// TIA Portal project "Project 3 Template_V15" (V15)

(* hardware
DEVICE "ET 200SP station_1"  ET 200SP-Station
   slot 0: "Rack_0"  Rack  6ES5 710-8MAx1
   slot 1: "PROJECT"  CPU 1512SP F-1 PN  6ES7 512-1SK01-0AB0  V1.8
   slot 2: "DC Input Card 1"  DI 8x24VDC HF  6ES7 131-6BF00-0CA0  V1.2
      slot 1: "DC Input Card 1"  DI 8x24VDC HF
   slot 3: "DC Input Card 2"  DI 8x24VDC HF  6ES7 131-6BF00-0CA0  V1.2
      slot 1: "DC Input Card 2"  DI 8x24VDC HF
   slot 4: "DC Output Card 1"  DQ 8x24VDC/0.5A HF  6ES7 132-6BF00-0CA0  V1.2
      slot 1: "DC Output Card 1"  DQ 8x24VDC/0.5A HF
   slot 5: "DC Output Card 2"  DQ 8x24VDC/0.5A HF  6ES7 132-6BF00-0CA0  V1.2
      slot 1: "DC Output Card 2"  DQ 8x24VDC/0.5A HF
   slot 6: "Analog Input Card 1"  AI 2xU/I 2,4-wire HS  6ES7 134-6HB00-0DA1  V1.1
      slot 1: "Analog Input Card 1"  AI 2xU/I 2,4-wire HS
   slot 7: "Analog Input Card 1_1"  AI 2xU/I 2,4-wire HS  6ES7 134-6HB00-0DA1  V1.1
      slot 1: "Analog Input Card 1_1"  AI 2xU/I 2,4-wire HS
   slot 8: "Analog Output Card"  AQ 2xU/I HS  6ES7 135-6HB00-0DA1  V1.1
      slot 1: "Analog Output Card"  AQ 2xU/I HS
   slot 9: "Server module_1"  Server module  6ES7 193-6PA00-0AA0  V1.0
      slot 1: "Server module_1"  Server module
   slot 127: "PROFINET BusAdapter CU"  BA 2xRJ45  6ES7 193-6AR00-0AA0  V0.0
      slot 32769: "Port_1"  6ES7 193-6AR00-0AA0
      slot 32770: "Port_2"  6ES7 193-6AR00-0AA0
DEVICE "GSD device_1"  GSD.Device.PN
   slot 0: "Rack"  Rail  V1.0
   slot 0: "WAGO"  750-377  V02.01.xx (03/04)
   slot 1: "75x-431 8DI_1"  75x-431
   slot 2: "75x-431 8DI_2"  75x-431
   slot 3: "75x-530(/0..-...) 8DO_1"  75x-530
   slot 4: "75x-530(/0..-...) 8DO_2"  75x-530
DEVICE "Visual Interface Simulator"  TP900 Comfort Portrait
   slot 0: "Visual Interface Simulator"  TP900 Comfort Portrait  6AV2 124-0JC01-0AX0  15.0.0.0
   slot 1: "HMI_RT_1"  TP900 Comfort Portrait  6AV2 124-0JC01-0AX0  15.0.0.0
   slot 5: "Visual Interface Simulator.IE_CP_1"  PROFINET Interface  15.0.0.0
      slot 1: "PROFINET Interface_1"  PROFINET Interface
         slot 1: "Port_1"  Port
         slot 2: "Port_2"  Port
   slot 7: "Visual Interface Simulator.MPI/DP_CP_1"  MPI/DP Interface  15.0.0.0
*)

// ===== PLC "PROJECT"  CPU 1512SP F-1 PN =====

VAR_GLOBAL   // PLC tag table "Default tag table"
   "Tag_1" AT %M1.0 : Bool;
   "INRange" AT %M1.4 : Bool;
   "Tag_3" AT %M13.1 : Bool;
   "Tag_4" AT %M9.0 : Bool;
   "Tag_6" AT %M7.1 : Bool;
   "FaultDetected" AT %M14.1 : Bool;
END_VAR

VAR_GLOBAL   // PLC tag table "R99_SIM Tags"
   "QB0" AT %QB0 : Byte;
   "IB0" AT %IB0 : Byte;
   "QB1" AT %QB1 : Byte;
   "QB70" AT %QB70 : Byte;
   "QB71" AT %QB71 : Byte;
   "IB1" AT %IB1 : Byte;
   "IB70" AT %IB70 : Byte;
   "IB71" AT %IB71 : Byte;
   "IW2" AT %IW2 : Int;
END_VAR

VAR_GLOBAL CONSTANT   // PLC tag table "R99_SIM Tags"
   "None(1)" : Pip := 65535;
   "Automatic update(1)" : Pip := 0;
   "PIP 1(1)" : Pip := 1;
   "PIP 2(1)" : Pip := 2;
   "PIP 3(1)" : Pip := 3;
   "PIP 4(1)" : Pip := 4;
   "PIP 5(1)" : Pip := 5;
   "PIP 6(1)" : Pip := 6;
   "PIP 7(1)" : Pip := 7;
   "PIP 8(1)" : Pip := 8;
   "PIP 9(1)" : Pip := 9;
   "PIP 10(1)" : Pip := 10;
   "PIP 11(1)" : Pip := 11;
   "PIP 12(1)" : Pip := 12;
   "PIP 13(1)" : Pip := 13;
   "PIP 14(1)" : Pip := 14;
   "PIP 15(1)" : Pip := 15;
   "PIP 16(1)" : Pip := 16;
   "PIP 17(1)" : Pip := 17;
   "PIP 18(1)" : Pip := 18;
   "PIP 19(1)" : Pip := 19;
   "PIP 20(1)" : Pip := 20;
   "PIP 21(1)" : Pip := 21;
   "PIP 22(1)" : Pip := 22;
   "PIP 23(1)" : Pip := 23;
   "PIP 24(1)" : Pip := 24;
   "PIP 25(1)" : Pip := 25;
   "PIP 26(1)" : Pip := 26;
   "PIP 27(1)" : Pip := 27;
   "PIP 28(1)" : Pip := 28;
   "PIP 29(1)" : Pip := 29;
   "PIP 30(1)" : Pip := 30;
   "PIP 31(1)" : Pip := 31;
   "PIP OB Servo(1)" : Pip := 32768;
   "Local~MC(1)" : Hw_SubModule := 51;
   "Local~Common(1)" : Hw_SubModule := 50;
   "Local~Device(1)" : Hw_Device := 32;
   "Local~Configuration(1)" : Hw_SubModule := 33;
   "Local~Exec(1)" : Hw_SubModule := 52;
   "Local(1)" : Hw_SubModule := 49;
   "Local~FExec(1)" : Hw_SubModule := 55;
   "Local~PROFINET_interface_1(1)" : Hw_Interface := 64;
   "Local~PROFINET_interface_1~Port_3(1)" : Hw_Interface := 67;
   "Local~PROFINET_interface_1~Port_1(1)" : Hw_Interface := 65;
   "Local~PROFINET_interface_1~Port_2(1)" : Hw_Interface := 66;
   "OB_Main(1)" : OB_PCYCLE := 1;
   "Local~DC_Input_Card_1_1(1)" : Hw_SubModule := 257;
   "Local~DC_Input_Card_2_1(1)" : Hw_SubModule := 258;
   "Local~DC_Output_Card_1_1(1)" : Hw_SubModule := 259;
   "Local~DC_Output_Card_2_1(1)" : Hw_SubModule := 260;
   "Local~Analog_Input_Card_1_1(1)" : Hw_SubModule := 261;
   "Local~Analog_Output_Card_1(1)" : Hw_SubModule := 263;
   "Local~Analog_Input_Card_1_1_2(1)" : Hw_SubModule := 262;
   "Local~PROFINET_IO-System(1)" : Hw_IoSystem := 264;
   "WAGO~Proxy(1)" : Hw_SubModule := 268;
   "WAGO~IODevice(1)" : Hw_Device := 266;
   "WAGO~Interface(1)" : Hw_Interface := 269;
   "WAGO~Interface~Port_1(1)" : Hw_Interface := 270;
   "WAGO~Interface~Port_2(1)" : Hw_Interface := 271;
   "WAGO~Head(1)" : Hw_SubModule := 272;
   "8DI~DI(2)" : Hw_SubModule := 273;
   "8DI~DI(3)" : Hw_SubModule := 274;
   "8DO~DO(2)" : Hw_SubModule := 275;
   "8DO~DO(3)" : Hw_SubModule := 276;
END_VAR

VAR_GLOBAL   // PLC tag table "project M File tag"
   "PNPExt" AT %Q70.0 : Bool;
   "PNPRet" AT %Q70.1 : Bool;
   "PNPRaise" AT %Q70.2 : Bool;
   "PNPlower" AT %Q70.3 : Bool;
   "PNPGrip" AT %Q70.4 : Bool;
   "ConEXT" AT %Q70.5 : Bool;
   "ConvRun" AT %Q70.6 : Bool;
   "extendPNP" AT %I70.0 : Bool;
   "retractPNP" AT %I70.1 : Bool;
   "raised" AT %I70.2 : Bool;
   "lower" AT %I70.3 : Bool;
   "Tag_5" AT %I70.4 : Bool;
   "convRet" AT %I70.5 : Bool;
   "partAtPickUp" AT %I70.6 : Bool;
   "StartPB" AT %I0.0 : Bool;
   "StopPB" AT %I0.1 : Bool;
   "PBA" AT %I0.2 : Bool;
   "PBB" AT %I0.3 : Bool;
   "SSA" AT %I0.4 : Bool;
   "MCR" AT %I0.5 : Bool;
   "EStopPB" AT %I0.6 : Bool;
   "GateSwitch" AT %I0.7 : Bool;
   "StartLight" AT %Q0.0 : Bool;
   "Tag_2" AT %Q0.1 : Bool;
   "LTA" AT %Q0.2 : Bool;
   "LTB" AT %Q0.3 : Bool;
END_VAR

TYPE "TPBool"
VERSION : 0.1
   STRUCT
      PB : Bool;
      LT : Bool;
   END_STRUCT;
END_TYPE

TYPE "TouchPanelPLC"
VERSION : 0.1
   STRUCT
      INT1 : Int;
      INT2 : Int;
      INT3 : Int;
      INT4 : Int;
      REAL1 : Real;
      REAL2 : Real;
      REAL3 : Real;
      REAL4 : Real;
      GRAY : "TPBool";
      BLUE : "TPBool";
      GREEN : "TPBool";
      YELLOW : "TPBool";
      RED : "TPBool";
   END_STRUCT;
END_TYPE

TYPE "TouchPanel"
VERSION : 0.1
   STRUCT
      PLC : "TouchPanelPLC";
      Stn : "TouchPanelStn";
      Conv : "TouchPanelConv";
   END_STRUCT;
END_TYPE

TYPE "TPExtRet"
VERSION : 0.1
   STRUCT
      Ext : "TPBool";
      Ret : "TPBool";
   END_STRUCT;
END_TYPE

TYPE "TPRaiseLower"
VERSION : 0.1
   STRUCT
      Raise : "TPBool";
      Lower : "TPBool";
   END_STRUCT;
END_TYPE

TYPE "TPOnOff"
VERSION : 0.1
   STRUCT
      On : "TPBool";
      Off : "TPBool";
   END_STRUCT;
END_TYPE

TYPE "TouchPanelStn"
VERSION : 0.1
   STRUCT
      Auto : "TPBool";
      Manual : "TPBool";
      CycleStart : "TPBool";
      CycleStop : "TPBool";
      Lift : "TPRaiseLower";
      PartRelease : "TPOnOff";
      Reject : "TPExtRet";
      Divert : "TPExtRet";
      SendToRejectChute : "TPBool";
      SendToDivertChute : "TPBool";
      SendToConv : "TPBool";
      InsertPart : "TPBool";
      FaultReset : "TPBool";
   END_STRUCT;
END_TYPE

TYPE "TouchPanelConv"
VERSION : 0.1
   STRUCT
      TargetSpeed : Real;
      Fwd : "TPBool";
      Rev : "TPBool";
      Stop : "TPBool";
      FaultReset : "TPBool";
      RemCntl : "TPOnOff";
   END_STRUCT;
END_TYPE

TYPE "SIM_CylinderAnimation"
VERSION : 0.1
   STRUCT
      Animation : DInt;
      Max : DInt;
      Extend : "SIM_Cylinder";
      Retract : "SIM_Cylinder";
   END_STRUCT;
END_TYPE

TYPE "SIM_Cylinder"
VERSION : 0.1
   STRUCT
      ScanCount : DInt;
      "Timer" : IEC_TIMER;
      Output : Bool;
      Sensor : Bool;
   END_STRUCT;
END_TYPE

TYPE "SIM_PLC"
VERSION : 0.1
   STRUCT
      IB0 : Byte;
      IB1 : Byte;
      IB70 : Byte;
      IB71 : Byte;
      QB0 : Byte;
      QB1 : Byte;
      QB70 : Byte;
      QB71 : Byte;
      PowerOnPB : Bool;
      Lift : "SIM_CylinderAnimation";
      Reject : "SIM_CylinderAnimation";
      Divert : "SIM_CylinderAnimation";
      "5sPulse" : IEC_TIMER;
      PartRelease : Bool;
      IW2 : Int;
      Oneshots : "Numbers";
      RandomTimer : IEC_TIMER;
      CH0RampUP : IEC_TIMER;
      CH0ACC : Int;
      RandomTime : Int;
      NewPartDelay : IEC_TIMER;
      PartClearDelay : IEC_TIMER;
   END_STRUCT;
END_TYPE

TYPE "Numbers"
VERSION : 0.1
   STRUCT
      "0" : Bool;
      "1" : Bool;
      "2" : Bool;
      "3" : Bool;
      "4" : Bool;
      "5" : Bool;
      "6" : Bool;
      "7" : Bool;
      "8" : Bool;
      "9" : Bool;
      "10" : Bool;
      "11" : Bool;
      "12" : Bool;
      "13" : Bool;
      "14" : Bool;
      "15" : Bool;
   END_STRUCT;
END_TYPE

DATA_BLOCK "TP"   // DB1
{ S7_Optimized_Access := 'FALSE' }
VERSION : 0.1
BEGIN
   PLC.GRAY.PB := true;
END_DATA_BLOCK

DATA_BLOCK "SIM"   // DB2
{ S7_Optimized_Access := 'FALSE' }
VERSION : 0.1
BEGIN
   IB0 := 2#10000010;
   Lift.Retract.Sensor := true;
   Reject.Retract.Sensor := true;
   Divert.Retract.Output := true;
   IB70 := 2#00000110;
END_DATA_BLOCK

DATA_BLOCK "project"   // DB3
{ S7_Optimized_Access := 'TRUE' }
VERSION : 0.1
   VAR
      RejectPartCount : Int;
      MaxWeight : Real;
      CycletimeREal : Real;
      cycletimeint : Int;
      PrevMaxWeight : Real;
      MaxWeigInt : Int;
   END_VAR
BEGIN
END_DATA_BLOCK

DATA_BLOCK "Project timers and counters"   // DB4
{ S7_Optimized_Access := 'TRUE' }
VERSION : 0.1
   VAR
      FaultTimer : IEC_TIMER;
      GoodPartCounters : IEC_COUNTER;
   END_VAR
   VAR RETAIN
      CycleTimer : IEC_TIMER;
   END_VAR
   VAR
      RetractionDelayTimer : IEC_TIMER;
      tptimer : IEC_TIMER;
      tofftimer : IEC_TIMER;
      extendGreenLt : IEC_TIMER;
   END_VAR
BEGIN
END_DATA_BLOCK

DATA_BLOCK "String Variables"   // DB12
{ S7_Optimized_Access := 'TRUE' }
VERSION : 0.1
   VAR RETAIN
      REAL1_TEXT : String := 'Real weight';
      REAL2_TEXT : String := 'curr weight';
      REAL3_TEXT : String := 'cycle time';
      REAL4_TEXT : String := 'Not used';
      INT1_TEXT : String := 'good part';
      INT2_TEXT : String := 'bad parts';
      INT3_TEXT : String := 'lower range';
      INT4_TEXT : String := 'higher range';
   END_VAR
BEGIN
END_DATA_BLOCK

FUNCTION "System Control" : Void   // FC1, LAD
{ S7_Optimized_Access := 'TRUE' }
VERSION : 0.1
// To Active cycle time, Press start PB , turn on MCR, the stop the it press PB
BEGIN

REGION Network 1
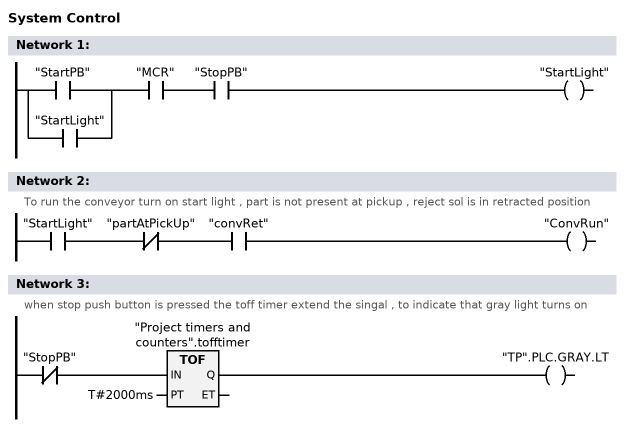
   RUNG wire#powerrail
      Contact( "StartPB" )
      wire#w1
      Contact( "MCR" )
      Contact( "StopPB" )
      Coil( "StartLight" )
   END_RUNG
   RUNG wire#powerrail
      Contact( "StartLight" )
   END_RUNG wire#w1
   // the same network as SCL:
   "StartLight" := ("StartPB" OR "StartLight") AND "MCR" AND "StopPB";
END_REGION

REGION Network 2
   // To run the conveyor turn on start light , part is not present at pickup , reject sol is in retracted position
   RUNG wire#powerrail
      Contact( "StartLight" )
      I_Contact( "partAtPickUp" )
      Contact( "convRet" )
      Coil( "ConvRun" )
   END_RUNG
   // the same network as SCL:
   "ConvRun" := "StartLight" AND NOT "partAtPickUp" AND "convRet";
END_REGION

REGION Network 3
   // when stop push button is pressed the toff timer extend the singal , to indicate that gray light turns on
   "Project timers and counters".tofftimer.TOF(IN := NOT "StopPB", PT := T#2000ms);
   "TP".PLC.GRAY.LT := "Project timers and counters".tofftimer.Q;
END_REGION
END_FUNCTION

FUNCTION "Weight Check Station Control" : Void   // FC2, LAD
{ S7_Optimized_Access := 'TRUE' }
VERSION : 0.1
   VAR_TEMP   // added for the SCL form of the ladder/FBD networks
      _w1 : Bool;
   END_VAR
BEGIN

REGION Network 1
   // To calculate the weight we need to convert the Analog value to the real weight in gms and displayed in real 1
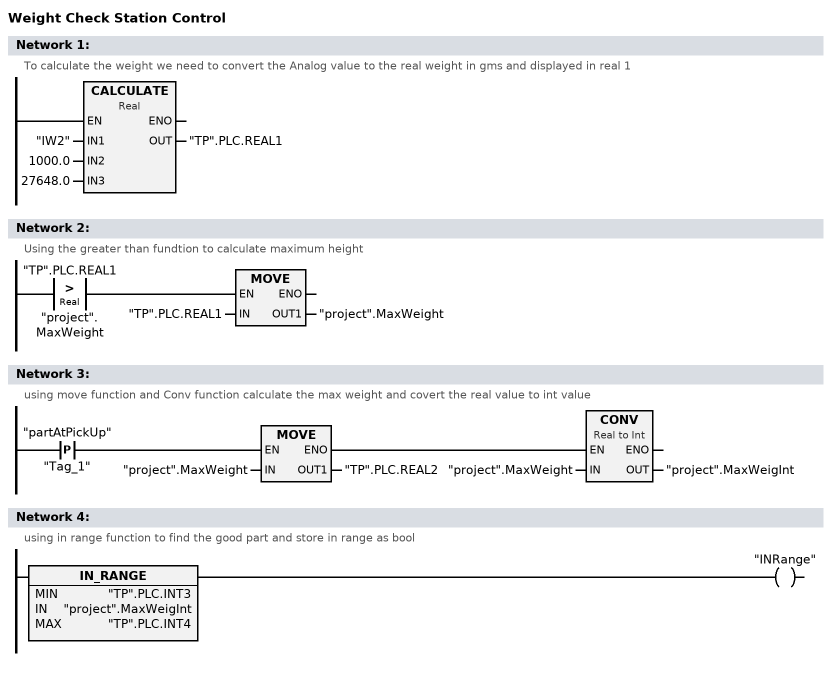
   RUNG wire#powerrail
      { S7_Templates := "SrcType := Real"; S7_Expression := "(IN2 / IN3) * IN1" } Calculate(in1 := "IW2", in2 := 1000.0, in3 := 27648.0, out => "TP".PLC.REAL1)
   END_RUNG
   // the same network as SCL:
   "TP".PLC.REAL1 := (1000.0 / 27648.0) * "IW2";
END_REGION

REGION Network 2
   // Using the greater than fundtion to calculate maximum height
   RUNG wire#powerrail
      { S7_Templates := "SrcType := Real" } GT_Contact(in1 := "TP".PLC.REAL1, in2 := "project".MaxWeight)
      Move(in := "TP".PLC.REAL1, out1 => "project".MaxWeight)
   END_RUNG
   // the same network as SCL:
   IF "TP".PLC.REAL1 > "project".MaxWeight THEN "project".MaxWeight := "TP".PLC.REAL1; END_IF;
END_REGION

REGION Network 3
   // using move function and Conv function calculate the max weight and covert the real value to int value
   RUNG wire#powerrail
      P_Contact(operand := "partAtPickUp", bit := "Tag_1")
      Move(in := "project".MaxWeight, out1 => "TP".PLC.REAL2)
      { S7_Templates := "[SrcType := Real, DestType := Int]" } Convert(in := "project".MaxWeight, out => "project".MaxWeigInt)
   END_RUNG
   // the same network as SCL:
   #_w1 := "partAtPickUp" AND NOT "Tag_1";   // rising edge of "partAtPickUp"
   "Tag_1" := "partAtPickUp";
   IF #_w1 THEN
       "TP".PLC.REAL2 := "project".MaxWeight;
       "project".MaxWeigInt := REAL_TO_INT("project".MaxWeight);
   END_IF;
END_REGION

REGION Network 4
   // using in range function to find the good part and store in range as bool
   RUNG wire#powerrail
      { S7_Templates := "SrcType := Int" } InRange(min := "TP".PLC.INT3, in := "project".MaxWeigInt, max := "TP".PLC.INT4)
      Coil( "INRange" )
   END_RUNG
   // the same network as SCL:
   "INRange" := ("TP".PLC.INT3 <= "project".MaxWeigInt) AND ("project".MaxWeigInt <= "TP".PLC.INT4);
END_REGION
END_FUNCTION

FUNCTION "Pick and Place Control" : Void   // FC3, LAD
{ S7_Optimized_Access := 'TRUE' }
VERSION : 0.1
BEGIN

REGION Network 1
   // To extedn reject sol , cycle time should be active , part is partpickup and value in not in range
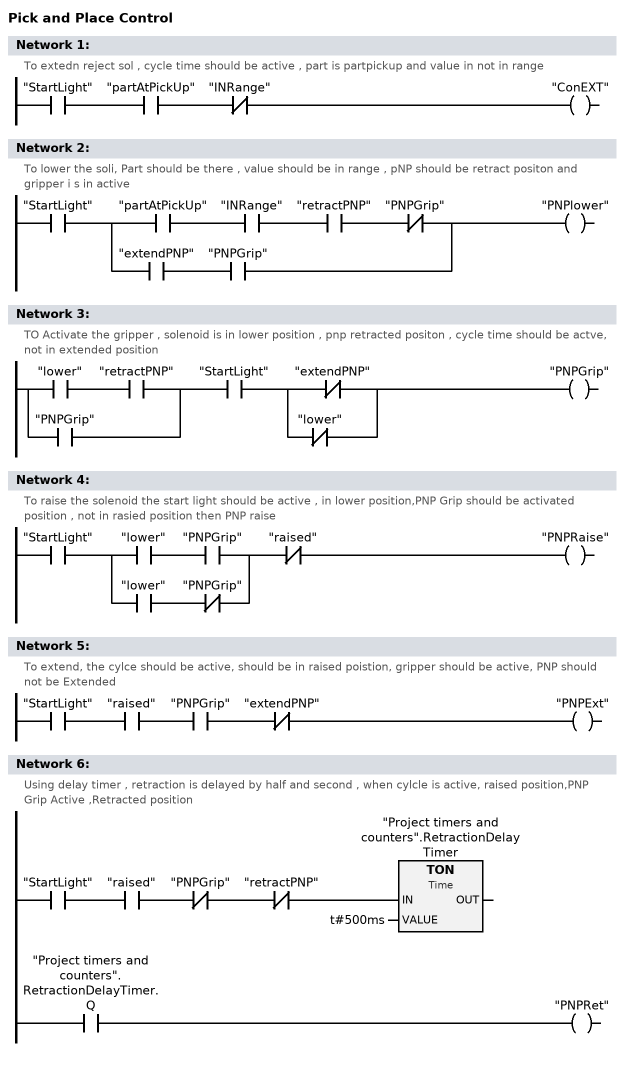
   RUNG wire#powerrail
      Contact( "StartLight" )
      Contact( "partAtPickUp" )
      I_Contact( "INRange" )
      Coil( "ConEXT" )
   END_RUNG
   // the same network as SCL:
   "ConEXT" := "StartLight" AND "partAtPickUp" AND NOT "INRange";
END_REGION

REGION Network 2
   // To lower the soli, Part should be there , value should be in range , pNP should be retract positon and gripper i s in active
   RUNG wire#powerrail
      Contact( "StartLight" )
      wire#w1
      Contact( "partAtPickUp" )
      Contact( "INRange" )
      Contact( "retractPNP" )
      I_Contact( "PNPGrip" )
      wire#w2
      Coil( "PNPlower" )
   END_RUNG
   RUNG wire#w1
      Contact( "extendPNP" )
      Contact( "PNPGrip" )
   END_RUNG wire#w2
   // the same network as SCL:
   "PNPlower" := "StartLight" AND (("partAtPickUp" AND "INRange" AND "retractPNP" AND NOT "PNPGrip") OR ("extendPNP" AND "PNPGrip"));
END_REGION

REGION Network 3
   // TO Activate the gripper , solenoid is in lower position , pnp retracted positon , cycle time should be actve, not in extended position
   RUNG wire#powerrail
      Contact( "lower" )
      Contact( "retractPNP" )
      wire#w1
      Contact( "StartLight" )
      wire#w2
      I_Contact( "extendPNP" )
      wire#w3
      Coil( "PNPGrip" )
   END_RUNG
   RUNG wire#powerrail
      Contact( "PNPGrip" )
   END_RUNG wire#w1
   RUNG wire#w2
      I_Contact( "lower" )
   END_RUNG wire#w3
   // the same network as SCL:
   "PNPGrip" := (("lower" AND "retractPNP") OR "PNPGrip") AND "StartLight" AND (NOT "extendPNP" OR NOT "lower");
END_REGION

REGION Network 4
   // To raise the solenoid the start light should be active , in lower position,PNP Grip should be activated position , not in rasied position then PNP raise
   RUNG wire#powerrail
      Contact( "StartLight" )
      wire#w1
      Contact( "lower" )
      Contact( "PNPGrip" )
      wire#w2
      I_Contact( "raised" )
      Coil( "PNPRaise" )
   END_RUNG
   RUNG wire#w1
      Contact( "lower" )
      I_Contact( "PNPGrip" )
   END_RUNG wire#w2
   // the same network as SCL:
   "PNPRaise" := "StartLight" AND (("lower" AND "PNPGrip") OR ("lower" AND NOT "PNPGrip")) AND NOT "raised";
END_REGION

REGION Network 5
   // To extend, the cylce should be active, should be in raised poistion, gripper should be active, PNP should not be Extended
   RUNG wire#powerrail
      Contact( "StartLight" )
      Contact( "raised" )
      Contact( "PNPGrip" )
      I_Contact( "extendPNP" )
      Coil( "PNPExt" )
   END_RUNG
   // the same network as SCL:
   "PNPExt" := "StartLight" AND "raised" AND "PNPGrip" AND NOT "extendPNP";
END_REGION

REGION Network 6
   // Using delay timer , retraction is delayed by half and second , when cylcle is active, raised position,PNP Grip Active ,Retracted position
   "Project timers and counters".RetractionDelayTimer.TON(IN := "StartLight" AND "raised" AND NOT "PNPGrip" AND NOT "retractPNP", PT := t#500ms);   // TON coil
   "PNPRet" := "Project timers and counters".RetractionDelayTimer.Q;
END_REGION
END_FUNCTION

FUNCTION "Faults" : Void   // FC4, LAD
{ S7_Optimized_Access := 'TRUE' }
VERSION : 0.1
BEGIN

REGION Network 1
   // using ton timer to find the faults , when extendion is not done in three seconds fault is detected
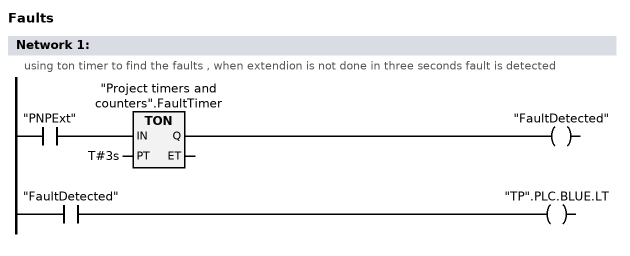
   "Project timers and counters".FaultTimer.TON(IN := "PNPExt", PT := T#3s);
   "FaultDetected" := "Project timers and counters".FaultTimer.Q;
   "TP".PLC.BLUE.LT := "FaultDetected";
END_REGION
END_FUNCTION

FUNCTION "Production Statistics" : Void   // FC5, LAD
{ S7_Optimized_Access := 'TRUE' }
VERSION : 0.1
   VAR_TEMP   // added for the SCL form of the ladder/FBD networks
      _w1 : Bool;
   END_VAR
BEGIN

REGION Network 1
   // Using a CTU counter instruction calculated the total number of good parts
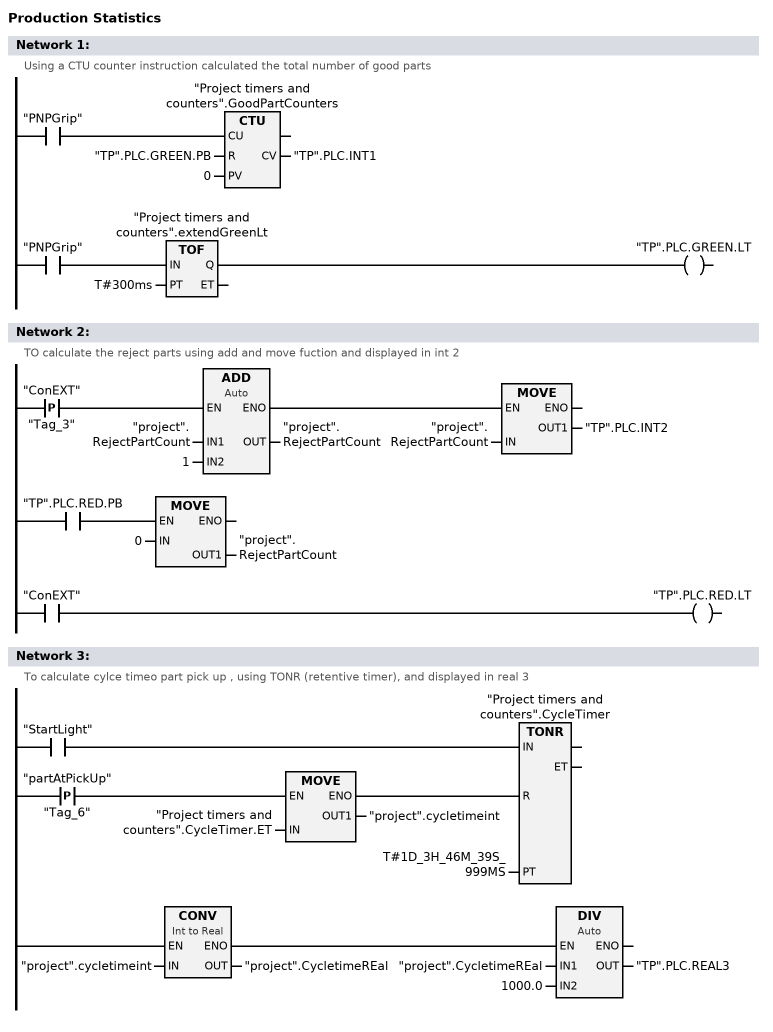
   "Project timers and counters".GoodPartCounters.CTU(CU := "PNPGrip",
                           R := "TP".PLC.GREEN.PB,
                           PV := 0,
                           CV => "TP".PLC.INT1);
   "Project timers and counters".extendGreenLt.TOF(IN := "PNPGrip", PT := T#300ms);
   "TP".PLC.GREEN.LT := "Project timers and counters".extendGreenLt.Q;
END_REGION

REGION Network 2
   // TO calculate the reject parts using add and move fuction and displayed in int 2
   RUNG wire#powerrail
      P_Contact(operand := "ConEXT", bit := "Tag_3")
      Add(in1 := "project".RejectPartCount, in2 := 1, out => "project".RejectPartCount)
      Move(in := "project".RejectPartCount, out1 => "TP".PLC.INT2)
   END_RUNG
   RUNG wire#powerrail
      Contact( "TP".PLC.RED.PB )
      Move(in := 0, out1 => "project".RejectPartCount)
   END_RUNG
   RUNG wire#powerrail
      Contact( "ConEXT" )
      Coil( "TP".PLC.RED.LT )
   END_RUNG
   // the same network as SCL:
   #_w1 := "ConEXT" AND NOT "Tag_3";   // rising edge of "ConEXT"
   "Tag_3" := "ConEXT";
   IF #_w1 THEN
       "project".RejectPartCount := "project".RejectPartCount + 1;
       "TP".PLC.INT2 := "project".RejectPartCount;
   END_IF;
   IF "TP".PLC.RED.PB THEN "project".RejectPartCount := 0; END_IF;
   "TP".PLC.RED.LT := "ConEXT";
END_REGION

REGION Network 3
   // To calculate cylce timeo part pick up , using TONR (retentive timer), and displayed in real 3
   #_w1 := "partAtPickUp" AND NOT "Tag_6";   // rising edge of "partAtPickUp"
   "Tag_6" := "partAtPickUp";
   IF #_w1 THEN "project".cycletimeint := "Project timers and counters".CycleTimer.ET; END_IF;
   "Project timers and counters".CycleTimer.TONR(IN := "StartLight", R := #_w1, PT := T#1D_3H_46M_39S_999MS);
   "project".CycletimeREal := INT_TO_REAL("project".cycletimeint);
   "TP".PLC.REAL3 := "project".CycletimeREal / 1000.0;
END_REGION
END_FUNCTION

FUNCTION "R99_Simulate" : Void   // FC99, LAD
{ S7_Optimized_Access := 'TRUE' }
VERSION : 0.1
   VAR_TEMP   // added for the SCL form of the ladder/FBD networks
      _w1 : Bool;
   END_VAR
BEGIN

REGION Network 1: Copy Outputs
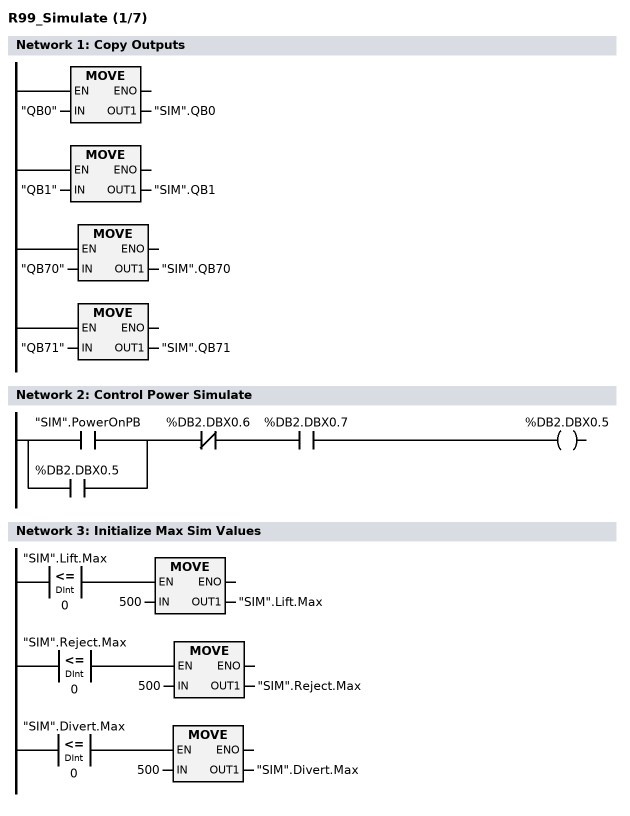
   RUNG wire#powerrail
      Move(in := "QB0", out1 => "SIM".QB0)
   END_RUNG
   RUNG wire#powerrail
      Move(in := "QB1", out1 => "SIM".QB1)
   END_RUNG
   RUNG wire#powerrail
      Move(in := "QB70", out1 => "SIM".QB70)
   END_RUNG
   RUNG wire#powerrail
      Move(in := "QB71", out1 => "SIM".QB71)
   END_RUNG
   // the same network as SCL:
   "SIM".QB0 := "QB0";
   "SIM".QB1 := "QB1";
   "SIM".QB70 := "QB70";
   "SIM".QB71 := "QB71";
END_REGION

REGION Network 2: Control Power Simulate
   RUNG wire#powerrail
      Contact( "SIM".PowerOnPB )
      wire#w1
      I_Contact( %DB2.DBX0.6 )
      Contact( %DB2.DBX0.7 )
      Coil( %DB2.DBX0.5 )
   END_RUNG
   RUNG wire#powerrail
      Contact( %DB2.DBX0.5 )
   END_RUNG wire#w1
   // the same network as SCL:
   %DB2.DBX0.5 := ("SIM".PowerOnPB OR %DB2.DBX0.5) AND NOT %DB2.DBX0.6 AND %DB2.DBX0.7;
END_REGION

REGION Network 3: Initialize Max Sim Values
   RUNG wire#powerrail
      { S7_Templates := "SrcType := DInt" } LE_Contact(in1 := "SIM".Lift.Max, in2 := 0)
      Move(in := 500, out1 => "SIM".Lift.Max)
   END_RUNG
   RUNG wire#powerrail
      { S7_Templates := "SrcType := DInt" } LE_Contact(in1 := "SIM".Reject.Max, in2 := 0)
      Move(in := 500, out1 => "SIM".Reject.Max)
   END_RUNG
   RUNG wire#powerrail
      { S7_Templates := "SrcType := DInt" } LE_Contact(in1 := "SIM".Divert.Max, in2 := 0)
      Move(in := 500, out1 => "SIM".Divert.Max)
   END_RUNG
   // the same network as SCL:
   IF "SIM".Lift.Max <= 0 THEN "SIM".Lift.Max := 500; END_IF;
   IF "SIM".Reject.Max <= 0 THEN "SIM".Reject.Max := 500; END_IF;
   IF "SIM".Divert.Max <= 0 THEN "SIM".Divert.Max := 500; END_IF;
END_REGION

REGION Network 4: Lift Simulate - Track Outputs
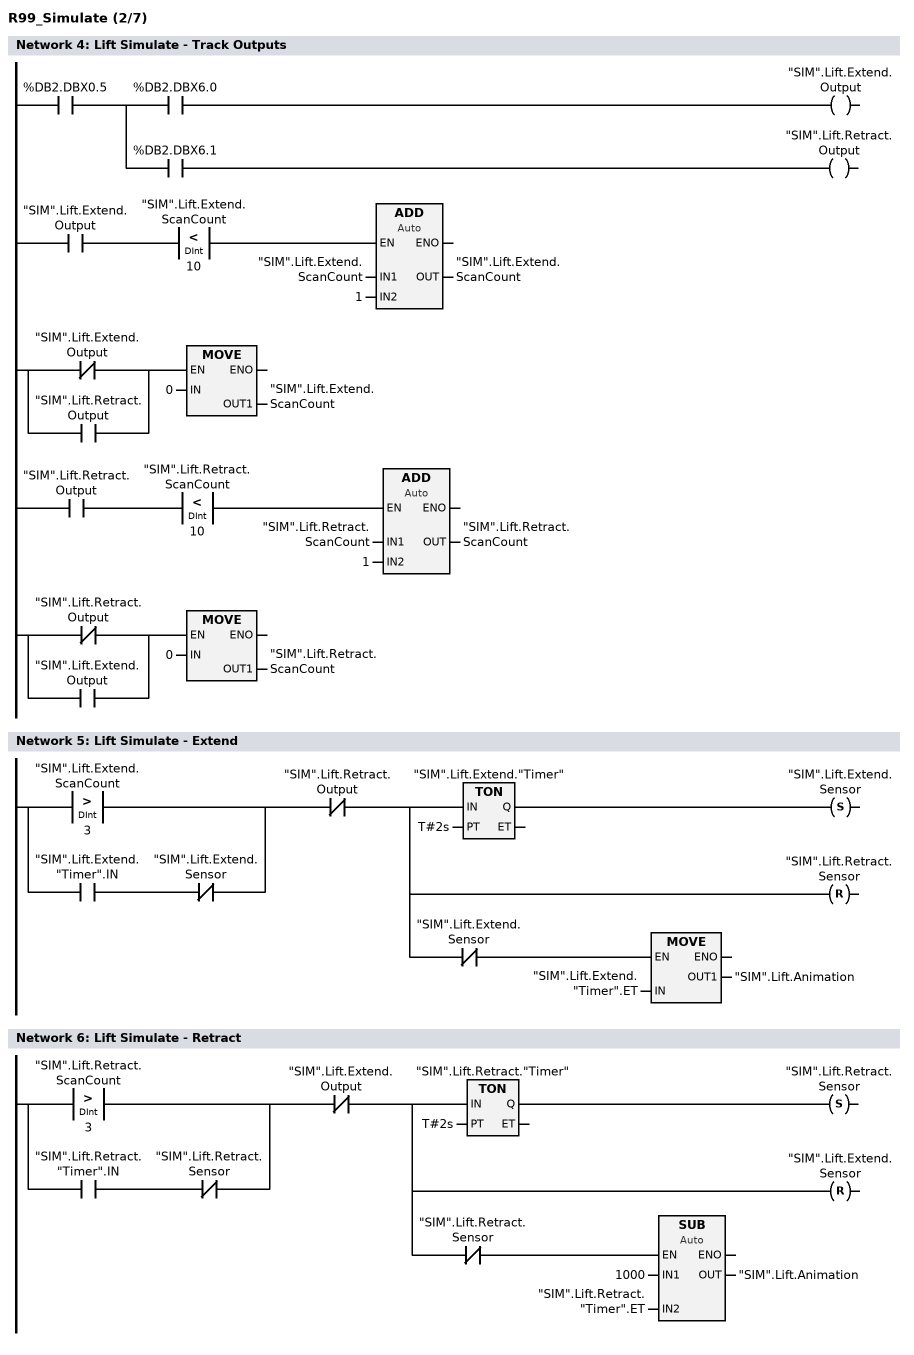
   RUNG wire#powerrail
      Contact( %DB2.DBX0.5 )
      wire#w1
      Contact( %DB2.DBX6.0 )
      Coil( "SIM".Lift.Extend.Output )
   END_RUNG
   RUNG wire#w1
      Contact( %DB2.DBX6.1 )
      Coil( "SIM".Lift.Retract.Output )
   END_RUNG
   RUNG wire#powerrail
      Contact( "SIM".Lift.Extend.Output )
      { S7_Templates := "SrcType := DInt" } LT_Contact(in1 := "SIM".Lift.Extend.ScanCount, in2 := 10)
      Add(in1 := "SIM".Lift.Extend.ScanCount, in2 := 1, out => "SIM".Lift.Extend.ScanCount)
   END_RUNG
   RUNG wire#powerrail
      I_Contact( "SIM".Lift.Extend.Output )
      wire#w2
      Move(in := 0, out1 => "SIM".Lift.Extend.ScanCount)
   END_RUNG
   RUNG wire#powerrail
      Contact( "SIM".Lift.Retract.Output )
   END_RUNG wire#w2
   RUNG wire#powerrail
      Contact( "SIM".Lift.Retract.Output )
      { S7_Templates := "SrcType := DInt" } LT_Contact(in1 := "SIM".Lift.Retract.ScanCount, in2 := 10)
      Add(in1 := "SIM".Lift.Retract.ScanCount, in2 := 1, out => "SIM".Lift.Retract.ScanCount)
   END_RUNG
   RUNG wire#powerrail
      I_Contact( "SIM".Lift.Retract.Output )
      wire#w3
      Move(in := 0, out1 => "SIM".Lift.Retract.ScanCount)
   END_RUNG
   RUNG wire#powerrail
      Contact( "SIM".Lift.Extend.Output )
   END_RUNG wire#w3
   // the same network as SCL:
   "SIM".Lift.Extend.Output := %DB2.DBX0.5 AND %DB2.DBX6.0;
   "SIM".Lift.Retract.Output := %DB2.DBX0.5 AND %DB2.DBX6.1;
   IF "SIM".Lift.Extend.Output AND ("SIM".Lift.Extend.ScanCount < 10) THEN
       "SIM".Lift.Extend.ScanCount := "SIM".Lift.Extend.ScanCount + 1;
   END_IF;
   IF NOT "SIM".Lift.Extend.Output OR "SIM".Lift.Retract.Output THEN
       "SIM".Lift.Extend.ScanCount := 0;
   END_IF;
   IF "SIM".Lift.Retract.Output AND ("SIM".Lift.Retract.ScanCount < 10) THEN
       "SIM".Lift.Retract.ScanCount := "SIM".Lift.Retract.ScanCount + 1;
   END_IF;
   IF NOT "SIM".Lift.Retract.Output OR "SIM".Lift.Extend.Output THEN
       "SIM".Lift.Retract.ScanCount := 0;
   END_IF;
END_REGION

REGION Network 5: Lift Simulate - Extend
   #_w1 := (("SIM".Lift.Extend.ScanCount > 3) OR ("SIM".Lift.Extend."Timer".IN AND NOT "SIM".Lift.Extend.Sensor)) AND NOT "SIM".Lift.Retract.Output;
   "SIM".Lift.Extend."Timer".TON(IN := #_w1, PT := T#2s);
   IF "SIM".Lift.Extend."Timer".Q THEN "SIM".Lift.Extend.Sensor := TRUE; END_IF;
   IF #_w1 THEN "SIM".Lift.Retract.Sensor := FALSE; END_IF;
   IF #_w1 AND NOT "SIM".Lift.Extend.Sensor THEN
       "SIM".Lift.Animation := "SIM".Lift.Extend."Timer".ET;
   END_IF;
END_REGION

REGION Network 6: Lift Simulate - Retract
   #_w1 := (("SIM".Lift.Retract.ScanCount > 3) OR ("SIM".Lift.Retract."Timer".IN AND NOT "SIM".Lift.Retract.Sensor)) AND NOT "SIM".Lift.Extend.Output;
   "SIM".Lift.Retract."Timer".TON(IN := #_w1, PT := T#2s);
   IF "SIM".Lift.Retract."Timer".Q THEN "SIM".Lift.Retract.Sensor := TRUE; END_IF;
   IF #_w1 THEN "SIM".Lift.Extend.Sensor := FALSE; END_IF;
   IF #_w1 AND NOT "SIM".Lift.Retract.Sensor THEN
       "SIM".Lift.Animation := 1000 - "SIM".Lift.Retract."Timer".ET;
   END_IF;
END_REGION

REGION Network 7: Lift Simulate - Update Sensors
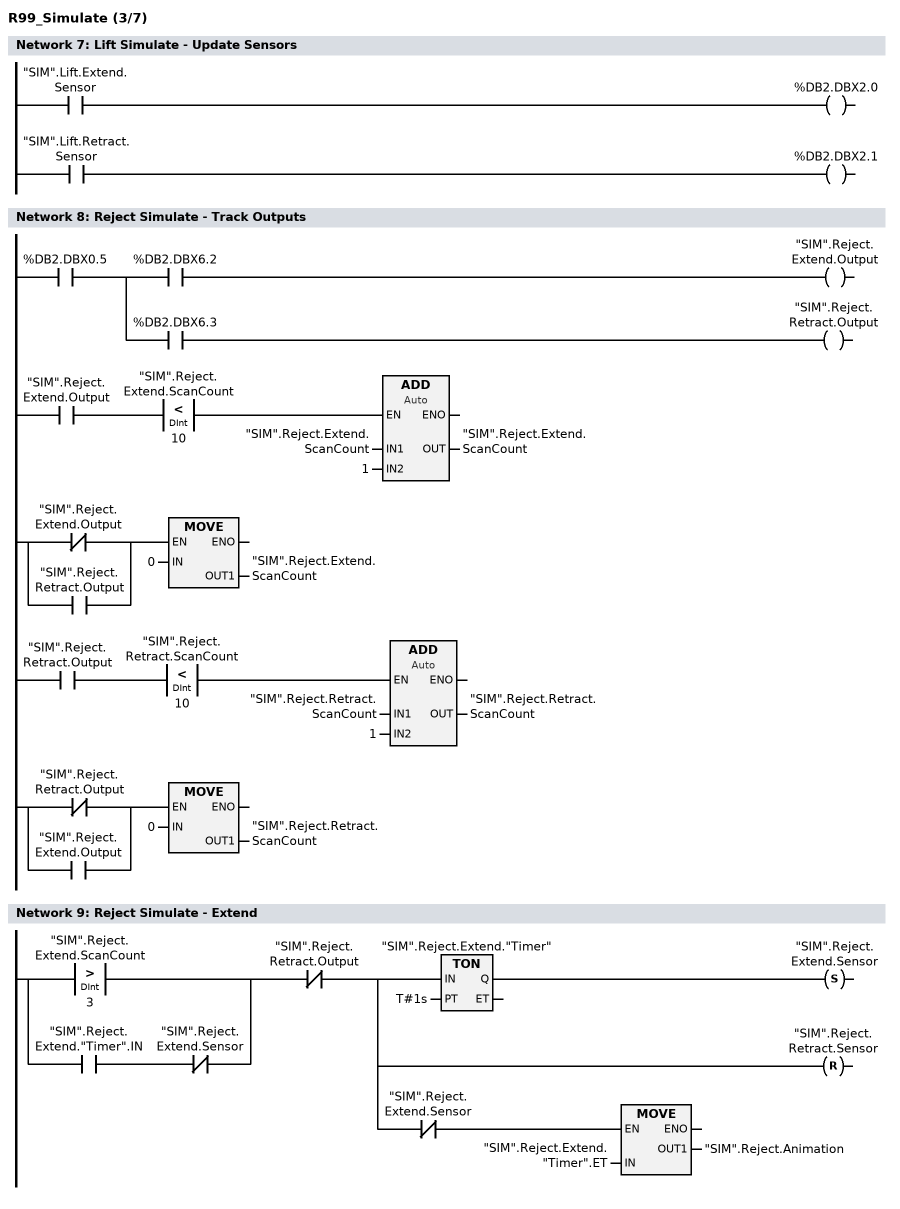
   RUNG wire#powerrail
      Contact( "SIM".Lift.Extend.Sensor )
      Coil( %DB2.DBX2.0 )
   END_RUNG
   RUNG wire#powerrail
      Contact( "SIM".Lift.Retract.Sensor )
      Coil( %DB2.DBX2.1 )
   END_RUNG
   // the same network as SCL:
   %DB2.DBX2.0 := "SIM".Lift.Extend.Sensor;
   %DB2.DBX2.1 := "SIM".Lift.Retract.Sensor;
END_REGION

REGION Network 8: Reject Simulate - Track Outputs
   RUNG wire#powerrail
      Contact( %DB2.DBX0.5 )
      wire#w1
      Contact( %DB2.DBX6.2 )
      Coil( "SIM".Reject.Extend.Output )
   END_RUNG
   RUNG wire#w1
      Contact( %DB2.DBX6.3 )
      Coil( "SIM".Reject.Retract.Output )
   END_RUNG
   RUNG wire#powerrail
      Contact( "SIM".Reject.Extend.Output )
      { S7_Templates := "SrcType := DInt" } LT_Contact(in1 := "SIM".Reject.Extend.ScanCount, in2 := 10)
      Add(in1 := "SIM".Reject.Extend.ScanCount, in2 := 1, out => "SIM".Reject.Extend.ScanCount)
   END_RUNG
   RUNG wire#powerrail
      I_Contact( "SIM".Reject.Extend.Output )
      wire#w2
      Move(in := 0, out1 => "SIM".Reject.Extend.ScanCount)
   END_RUNG
   RUNG wire#powerrail
      Contact( "SIM".Reject.Retract.Output )
   END_RUNG wire#w2
   RUNG wire#powerrail
      Contact( "SIM".Reject.Retract.Output )
      { S7_Templates := "SrcType := DInt" } LT_Contact(in1 := "SIM".Reject.Retract.ScanCount, in2 := 10)
      Add(in1 := "SIM".Reject.Retract.ScanCount, in2 := 1, out => "SIM".Reject.Retract.ScanCount)
   END_RUNG
   RUNG wire#powerrail
      I_Contact( "SIM".Reject.Retract.Output )
      wire#w3
      Move(in := 0, out1 => "SIM".Reject.Retract.ScanCount)
   END_RUNG
   RUNG wire#powerrail
      Contact( "SIM".Reject.Extend.Output )
   END_RUNG wire#w3
   // the same network as SCL:
   "SIM".Reject.Extend.Output := %DB2.DBX0.5 AND %DB2.DBX6.2;
   "SIM".Reject.Retract.Output := %DB2.DBX0.5 AND %DB2.DBX6.3;
   IF "SIM".Reject.Extend.Output AND ("SIM".Reject.Extend.ScanCount < 10) THEN
       "SIM".Reject.Extend.ScanCount := "SIM".Reject.Extend.ScanCount + 1;
   END_IF;
   IF NOT "SIM".Reject.Extend.Output OR "SIM".Reject.Retract.Output THEN
       "SIM".Reject.Extend.ScanCount := 0;
   END_IF;
   IF "SIM".Reject.Retract.Output AND ("SIM".Reject.Retract.ScanCount < 10) THEN
       "SIM".Reject.Retract.ScanCount := "SIM".Reject.Retract.ScanCount + 1;
   END_IF;
   IF NOT "SIM".Reject.Retract.Output OR "SIM".Reject.Extend.Output THEN
       "SIM".Reject.Retract.ScanCount := 0;
   END_IF;
END_REGION

REGION Network 9: Reject Simulate - Extend
   #_w1 := (("SIM".Reject.Extend.ScanCount > 3) OR ("SIM".Reject.Extend."Timer".IN AND NOT "SIM".Reject.Extend.Sensor)) AND NOT "SIM".Reject.Retract.Output;
   "SIM".Reject.Extend."Timer".TON(IN := #_w1, PT := T#1s);
   IF "SIM".Reject.Extend."Timer".Q THEN "SIM".Reject.Extend.Sensor := TRUE; END_IF;
   IF #_w1 THEN "SIM".Reject.Retract.Sensor := FALSE; END_IF;
   IF #_w1 AND NOT "SIM".Reject.Extend.Sensor THEN
       "SIM".Reject.Animation := "SIM".Reject.Extend."Timer".ET;
   END_IF;
END_REGION

REGION Network 10: Reject Simulate - Retract
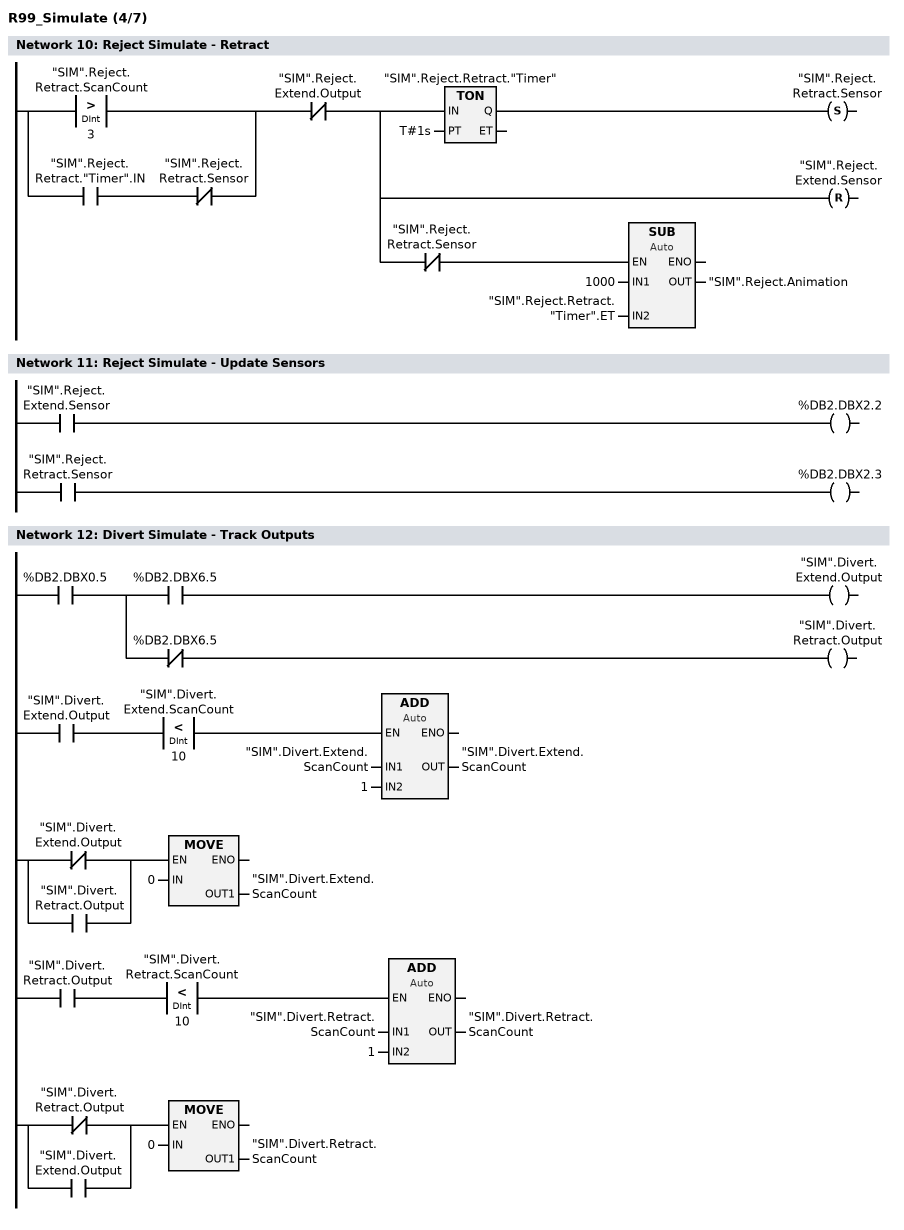
   #_w1 := (("SIM".Reject.Retract.ScanCount > 3) OR ("SIM".Reject.Retract."Timer".IN AND NOT "SIM".Reject.Retract.Sensor)) AND NOT "SIM".Reject.Extend.Output;
   "SIM".Reject.Retract."Timer".TON(IN := #_w1, PT := T#1s);
   IF "SIM".Reject.Retract."Timer".Q THEN "SIM".Reject.Retract.Sensor := TRUE; END_IF;
   IF #_w1 THEN "SIM".Reject.Extend.Sensor := FALSE; END_IF;
   IF #_w1 AND NOT "SIM".Reject.Retract.Sensor THEN
       "SIM".Reject.Animation := 1000 - "SIM".Reject.Retract."Timer".ET;
   END_IF;
END_REGION

REGION Network 11: Reject Simulate - Update Sensors
   RUNG wire#powerrail
      Contact( "SIM".Reject.Extend.Sensor )
      Coil( %DB2.DBX2.2 )
   END_RUNG
   RUNG wire#powerrail
      Contact( "SIM".Reject.Retract.Sensor )
      Coil( %DB2.DBX2.3 )
   END_RUNG
   // the same network as SCL:
   %DB2.DBX2.2 := "SIM".Reject.Extend.Sensor;
   %DB2.DBX2.3 := "SIM".Reject.Retract.Sensor;
END_REGION

REGION Network 12: Divert Simulate - Track Outputs
   RUNG wire#powerrail
      Contact( %DB2.DBX0.5 )
      wire#w1
      Contact( %DB2.DBX6.5 )
      Coil( "SIM".Divert.Extend.Output )
   END_RUNG
   RUNG wire#w1
      I_Contact( %DB2.DBX6.5 )
      Coil( "SIM".Divert.Retract.Output )
   END_RUNG
   RUNG wire#powerrail
      Contact( "SIM".Divert.Extend.Output )
      { S7_Templates := "SrcType := DInt" } LT_Contact(in1 := "SIM".Divert.Extend.ScanCount, in2 := 10)
      Add(in1 := "SIM".Divert.Extend.ScanCount, in2 := 1, out => "SIM".Divert.Extend.ScanCount)
   END_RUNG
   RUNG wire#powerrail
      I_Contact( "SIM".Divert.Extend.Output )
      wire#w2
      Move(in := 0, out1 => "SIM".Divert.Extend.ScanCount)
   END_RUNG
   RUNG wire#powerrail
      Contact( "SIM".Divert.Retract.Output )
   END_RUNG wire#w2
   RUNG wire#powerrail
      Contact( "SIM".Divert.Retract.Output )
      { S7_Templates := "SrcType := DInt" } LT_Contact(in1 := "SIM".Divert.Retract.ScanCount, in2 := 10)
      Add(in1 := "SIM".Divert.Retract.ScanCount, in2 := 1, out => "SIM".Divert.Retract.ScanCount)
   END_RUNG
   RUNG wire#powerrail
      I_Contact( "SIM".Divert.Retract.Output )
      wire#w3
      Move(in := 0, out1 => "SIM".Divert.Retract.ScanCount)
   END_RUNG
   RUNG wire#powerrail
      Contact( "SIM".Divert.Extend.Output )
   END_RUNG wire#w3
   // the same network as SCL:
   "SIM".Divert.Extend.Output := %DB2.DBX0.5 AND %DB2.DBX6.5;
   "SIM".Divert.Retract.Output := %DB2.DBX0.5 AND NOT %DB2.DBX6.5;
   IF "SIM".Divert.Extend.Output AND ("SIM".Divert.Extend.ScanCount < 10) THEN
       "SIM".Divert.Extend.ScanCount := "SIM".Divert.Extend.ScanCount + 1;
   END_IF;
   IF NOT "SIM".Divert.Extend.Output OR "SIM".Divert.Retract.Output THEN
       "SIM".Divert.Extend.ScanCount := 0;
   END_IF;
   IF "SIM".Divert.Retract.Output AND ("SIM".Divert.Retract.ScanCount < 10) THEN
       "SIM".Divert.Retract.ScanCount := "SIM".Divert.Retract.ScanCount + 1;
   END_IF;
   IF NOT "SIM".Divert.Retract.Output OR "SIM".Divert.Extend.Output THEN
       "SIM".Divert.Retract.ScanCount := 0;
   END_IF;
END_REGION

REGION Network 13: Divert Simulate - Extend
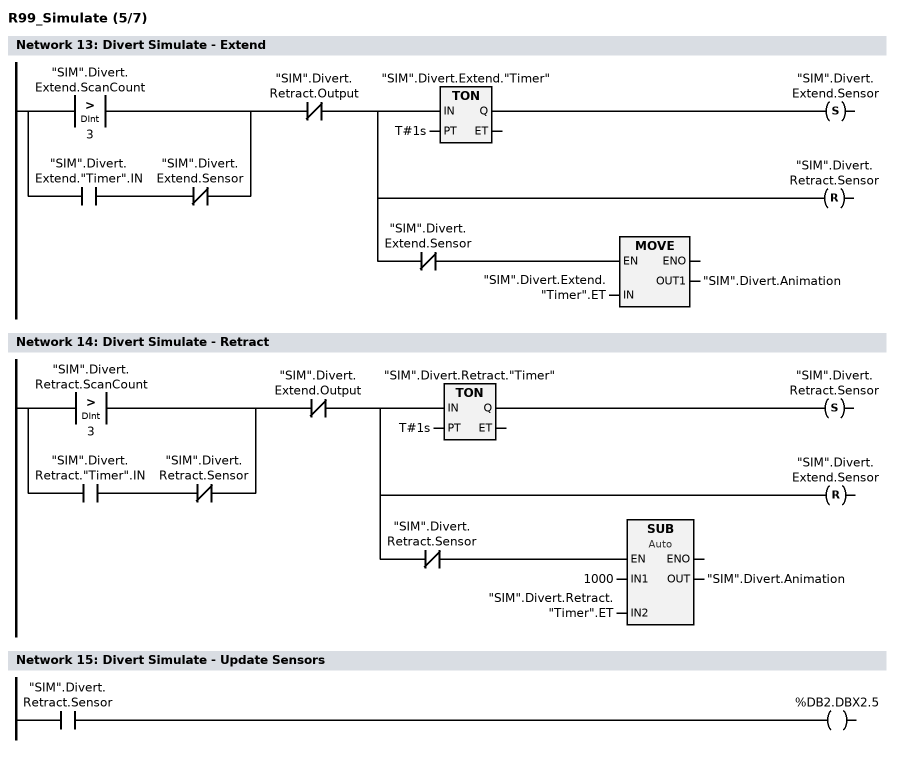
   #_w1 := (("SIM".Divert.Extend.ScanCount > 3) OR ("SIM".Divert.Extend."Timer".IN AND NOT "SIM".Divert.Extend.Sensor)) AND NOT "SIM".Divert.Retract.Output;
   "SIM".Divert.Extend."Timer".TON(IN := #_w1, PT := T#1s);
   IF "SIM".Divert.Extend."Timer".Q THEN "SIM".Divert.Extend.Sensor := TRUE; END_IF;
   IF #_w1 THEN "SIM".Divert.Retract.Sensor := FALSE; END_IF;
   IF #_w1 AND NOT "SIM".Divert.Extend.Sensor THEN
       "SIM".Divert.Animation := "SIM".Divert.Extend."Timer".ET;
   END_IF;
END_REGION

REGION Network 14: Divert Simulate - Retract
   #_w1 := (("SIM".Divert.Retract.ScanCount > 3) OR ("SIM".Divert.Retract."Timer".IN AND NOT "SIM".Divert.Retract.Sensor)) AND NOT "SIM".Divert.Extend.Output;
   "SIM".Divert.Retract."Timer".TON(IN := #_w1, PT := T#1s);
   IF "SIM".Divert.Retract."Timer".Q THEN "SIM".Divert.Retract.Sensor := TRUE; END_IF;
   IF #_w1 THEN "SIM".Divert.Extend.Sensor := FALSE; END_IF;
   IF #_w1 AND NOT "SIM".Divert.Retract.Sensor THEN
       "SIM".Divert.Animation := 1000 - "SIM".Divert.Retract."Timer".ET;
   END_IF;
END_REGION

REGION Network 15: Divert Simulate - Update Sensors
   RUNG wire#powerrail
      Contact( "SIM".Divert.Retract.Sensor )
      Coil( %DB2.DBX2.5 )
   END_RUNG
   // the same network as SCL:
   %DB2.DBX2.5 := "SIM".Divert.Retract.Sensor;
END_REGION

REGION Network 16: Simulate Analog Sensor
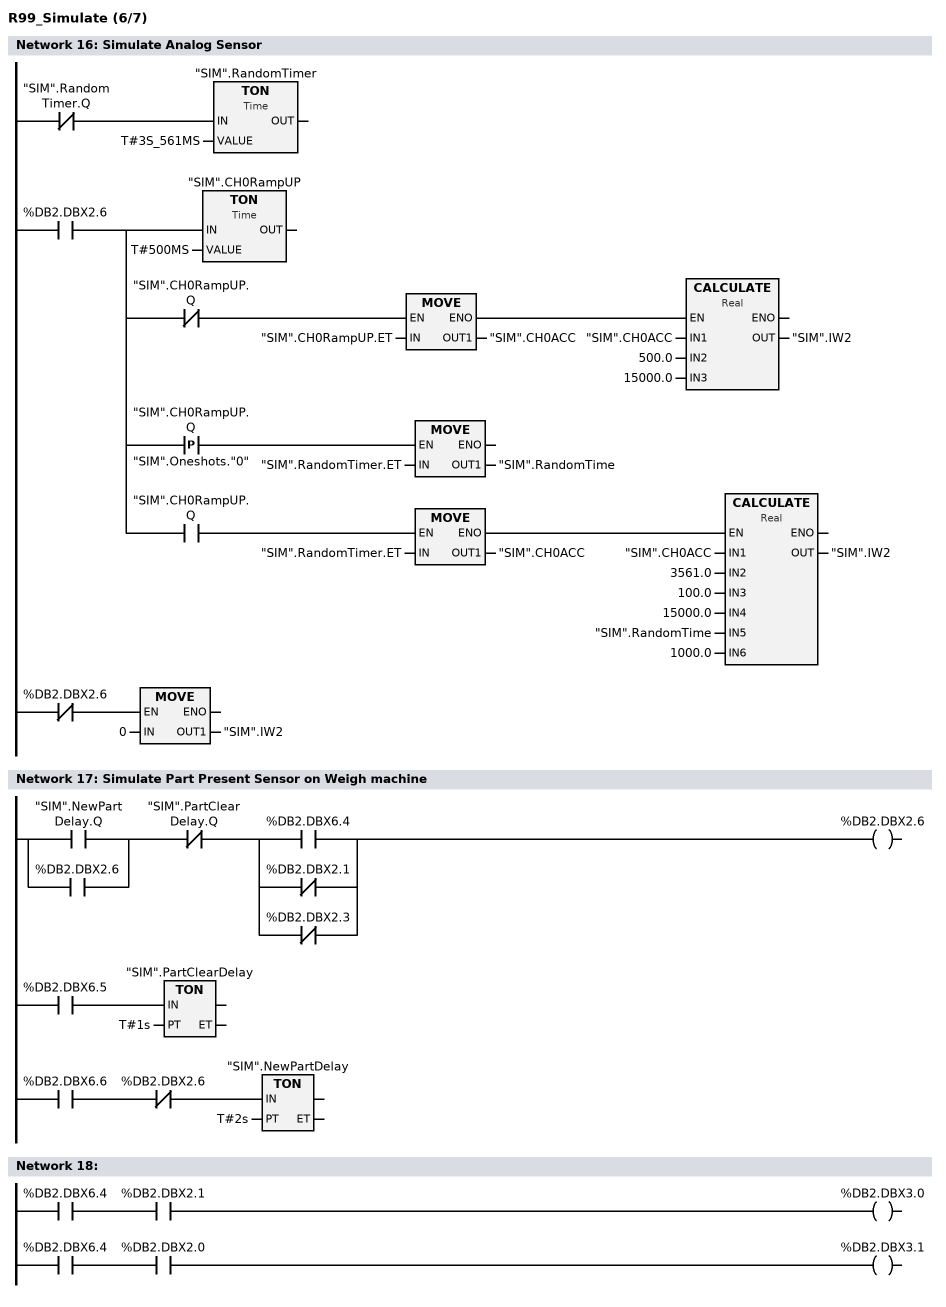
   "SIM".RandomTimer.TON(IN := NOT "SIM".RandomTimer.Q, PT := T#3S_561MS);   // TON coil
   "SIM".CH0RampUP.TON(IN := %DB2.DBX2.6, PT := T#500MS);   // TON coil
   IF %DB2.DBX2.6 AND NOT "SIM".CH0RampUP.Q THEN
       "SIM".CH0ACC := "SIM".CH0RampUP.ET;
       "SIM".IW2 := "SIM".CH0ACC/500.0*15000.0;
   END_IF;
   #_w1 := %DB2.DBX2.6 AND "SIM".CH0RampUP.Q AND NOT "SIM".Oneshots."0";   // rising edge of "SIM".CH0RampUP.Q
   "SIM".Oneshots."0" := "SIM".CH0RampUP.Q;
   IF #_w1 THEN "SIM".RandomTime := "SIM".RandomTimer.ET; END_IF;
   IF %DB2.DBX2.6 AND "SIM".CH0RampUP.Q THEN
       "SIM".CH0ACC := "SIM".RandomTimer.ET;
       "SIM".IW2 := "SIM".CH0ACC/3561.0*100.0+"SIM".RandomTime/3561.0*1000.0+15000.0;
   END_IF;
   IF NOT %DB2.DBX2.6 THEN "SIM".IW2 := 0; END_IF;
END_REGION

REGION Network 17: Simulate Part Present Sensor on Weigh machine
   %DB2.DBX2.6 := ("SIM".NewPartDelay.Q OR %DB2.DBX2.6) AND NOT "SIM".PartClearDelay.Q AND (%DB2.DBX6.4 OR NOT %DB2.DBX2.1 OR NOT %DB2.DBX2.3);
   "SIM".PartClearDelay.TON(IN := %DB2.DBX6.5, PT := T#1s);
   "SIM".NewPartDelay.TON(IN := %DB2.DBX6.6 AND NOT %DB2.DBX2.6, PT := T#2s);
END_REGION

REGION Network 18
   RUNG wire#powerrail
      Contact( %DB2.DBX6.4 )
      Contact( %DB2.DBX2.1 )
      Coil( %DB2.DBX3.0 )
   END_RUNG
   RUNG wire#powerrail
      Contact( %DB2.DBX6.4 )
      Contact( %DB2.DBX2.0 )
      Coil( %DB2.DBX3.1 )
   END_RUNG
   // the same network as SCL:
   %DB2.DBX3.0 := %DB2.DBX6.4 AND %DB2.DBX2.1;
   %DB2.DBX3.1 := %DB2.DBX6.4 AND %DB2.DBX2.0;
END_REGION

REGION Network 19: Copy Inputs
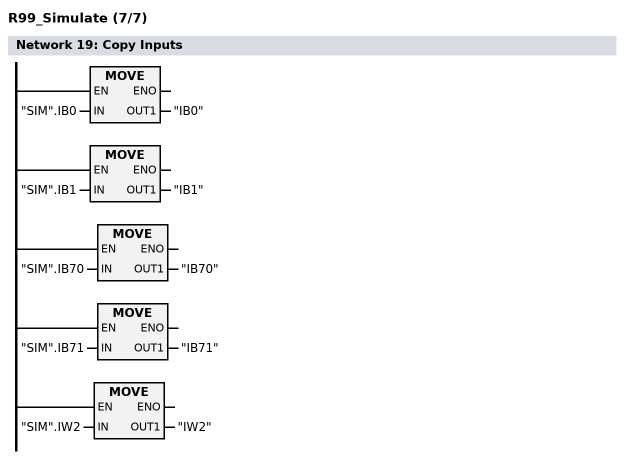
   RUNG wire#powerrail
      Move(in := "SIM".IB0, out1 => "IB0")
   END_RUNG
   RUNG wire#powerrail
      Move(in := "SIM".IB1, out1 => "IB1")
   END_RUNG
   RUNG wire#powerrail
      Move(in := "SIM".IB70, out1 => "IB70")
   END_RUNG
   RUNG wire#powerrail
      Move(in := "SIM".IB71, out1 => "IB71")
   END_RUNG
   RUNG wire#powerrail
      Move(in := "SIM".IW2, out1 => "IW2")
   END_RUNG
   // the same network as SCL:
   "IB0" := "SIM".IB0;
   "IB1" := "SIM".IB1;
   "IB70" := "SIM".IB70;
   "IB71" := "SIM".IB71;
   "IW2" := "SIM".IW2;
END_REGION
END_FUNCTION

ORGANIZATION_BLOCK "Main"   // OB1, LAD, ProgramCycle
TITLE = "Main Program Sweep (Cycle)"
{ S7_Optimized_Access := 'TRUE' }
VERSION : 0.1
   VAR_INPUT
      Initial_Call : Bool;   // Initial call of this OB
      Remanence : Bool;   // =True, if remanent data are available
   END_VAR
BEGIN

REGION Network 1: SIMULATE LOGIC - DO NOT CHANGE
   // Make sure this is always Network 1 and do not add anything else to this rung.
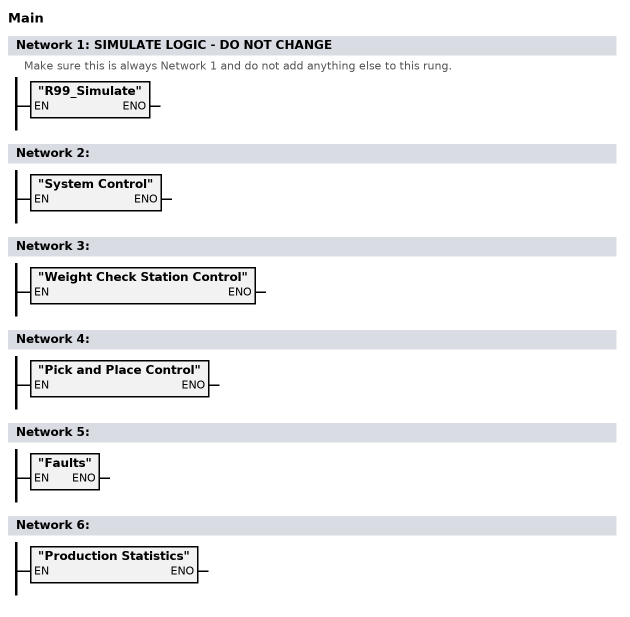
   RUNG wire#powerrail
      "R99_Simulate"()
   END_RUNG
   // the same network as SCL:
   "R99_Simulate"();
END_REGION

REGION Network 2
   RUNG wire#powerrail
      "System Control"()
   END_RUNG
   // the same network as SCL:
   "System Control"();
END_REGION

REGION Network 3
   RUNG wire#powerrail
      "Weight Check Station Control"()
   END_RUNG
   // the same network as SCL:
   "Weight Check Station Control"();
END_REGION

REGION Network 4
   RUNG wire#powerrail
      "Pick and Place Control"()
   END_RUNG
   // the same network as SCL:
   "Pick and Place Control"();
END_REGION

REGION Network 5
   RUNG wire#powerrail
      "Faults"()
   END_RUNG
   // the same network as SCL:
   "Faults"();
END_REGION

REGION Network 6
   RUNG wire#powerrail
      "Production Statistics"()
   END_RUNG
   // the same network as SCL:
   "Production Statistics"();
END_REGION
END_ORGANIZATION_BLOCK

(* ===== HMI "HMI_RT_1" =====
system functions are stored by id; their names below are inferred from use
connection "SIPLC": ETHERNET, S7_1500_OMS
connection "HMI_Connection_1": ETHERNET, S7_1500_OMS

HMI tags "Default tag table"
   "Station" : Int, internal

HMI tags "SIEMENS PLC Tags"
   "SIEMENS GREENLT" : Bool AT %DB1.DBX28.1, 100 ms
   "SIEMENS REAL2" : Real AT %DB1.DBD12, 100 ms
   "SIEMENS INT2" : Int AT %DB1.DBW2, 100 ms
   "SIEMENS YELLOWPB" : Bool AT %DB1.DBX30.0, 100 ms
   "SIEMENS REAL4" : Real AT %DB1.DBD20, 100 ms
   "SIEMENS REDLT" : Bool AT %DB1.DBX32.1, 100 ms
   "SIEMENS CH0" : Int AT %DB2.DBW184, 100 ms
   "SIEMENS INPUTS" : Byte AT %IB1, 100 ms
   "SIEMENS REAL3" : Real AT %DB1.DBD16, 100 ms
   "SIEMENS BLUELT" : Bool AT %DB1.DBX26.1, 100 ms
   "SIEMENS YELLOWLT" : Bool AT %DB1.DBX30.1, 100 ms
   "SIEMENS GRAYPB" : Bool AT %DB1.DBX24.0, 100 ms
   "SIEMENS BLUEPB" : Bool AT %DB1.DBX26.0, 100 ms
   "SIEMENS CH1" : Int AT %IW4, 100 ms
   "SIEMENS GRAYLT" : Bool AT %DB1.DBX24.1, 100 ms
   "SIEMENS GREENPB" : Bool AT %DB1.DBX28.0, 100 ms
   "SIEMENS INT1" : Int AT %DB1.DBW0, 100 ms
   "SIEMENS REDPB" : Bool AT %DB1.DBX32.0, 100 ms
   "SIEMENS INT3" : Int AT %DB1.DBW4, 100 ms
   "SIEMENS REAL1" : Real AT %DB1.DBD8, 100 ms
   "SIEMENS INT4" : Int AT %DB1.DBW6, 100 ms
   "SIEMENS NINA DATA" : Byte AT %IB70, 100 ms
   "SIEMENS NINB DATA" : Byte AT %IB71, 100 ms
   "SIEMENS LINA DATA" : Byte AT %IB0, 100 ms
   "SIEMENS LINB DATA" : Byte AT %IB1, 100 ms
   "SIEMENS LOUTA DATA" : Byte AT %QB0, 100 ms
   "SIEMENS LOUTB DATA" : Byte AT %QB1, 100 ms
   "SIEMENS NOUTA DATA" : Byte AT %QB70, 100 ms
   "SIEMENS NOUTB DATA" : Byte AT %QB71, 100 ms
   "SIEMENS CHQ0" : Int AT %QW2, 100 ms

HMI tags "SIEMENS IO Tags"
   "I0_0" : Bool AT %DB2.DBX0.0, 100 ms
   "I0_1" : Bool AT %DB2.DBX0.1, 100 ms
   "I0_2" : Bool AT %DB2.DBX0.2, 100 ms
   "I0_3" : Bool AT %DB2.DBX0.3, 100 ms
   "I0_4" : Bool AT %DB2.DBX0.4, 100 ms
   "I0_5" : Bool AT %DB2.DBX0.5, 100 ms
   "I0_6" : Bool AT %DB2.DBX0.6, 100 ms
   "I0_7" : Bool AT %DB2.DBX0.7, 100 ms
   "I1_0" : Bool AT %DB2.DBX1.0, 100 ms
   "I1_1" : Bool AT %DB2.DBX1.1, 100 ms
   "I1_2" : Bool AT %DB2.DBX1.2, 100 ms
   "I1_3" : Bool AT %DB2.DBX1.3, 100 ms
   "I1_4" : Bool AT %DB2.DBX1.4, 100 ms
   "I1_5" : Bool AT %DB2.DBX1.5, 100 ms
   "I1_6" : Bool AT %DB2.DBX1.6, 100 ms
   "I1_7" : Bool AT %DB2.DBX1.7, 100 ms
   "I70_0" : Bool AT %DB2.DBX2.0, 100 ms
   "I70_1" : Bool AT %DB2.DBX2.1, 100 ms
   "I70_2" : Bool AT %DB2.DBX2.2, 100 ms
   "I70_3" : Bool AT %DB2.DBX2.3, 100 ms
   "I70_4" : Bool AT %DB2.DBX2.4, 100 ms
   "I70_5" : Bool AT %DB2.DBX2.5, 100 ms
   "I70_6" : Bool AT %DB2.DBX2.6, 100 ms
   "I70_7" : Bool AT %DB2.DBX2.7, 100 ms
   "I71_0" : Bool AT %DB2.DBX3.0, 100 ms
   "I71_1" : Bool AT %DB2.DBX3.1, 100 ms
   "I71_2" : Bool AT %DB2.DBX3.2, 100 ms
   "I71_3" : Bool AT %DB2.DBX3.3, 100 ms
   "I71_4" : Bool AT %DB2.DBX3.4, 100 ms
   "I71_5" : Bool AT %DB2.DBX3.5, 100 ms
   "I71_6" : Bool AT %DB2.DBX3.6, 100 ms
   "I71_7" : Bool AT %DB2.DBX3.7, 100 ms
   "Q0_0" : Bool AT %DB2.DBX4.0, 100 ms
   "Q0_1" : Bool AT %DB2.DBX4.1, 100 ms
   "Q0_2" : Bool AT %DB2.DBX4.2, 100 ms
   "Q0_3" : Bool AT %DB2.DBX4.3, 100 ms
   "Q0_4" : Bool AT %DB2.DBX4.4, 100 ms
   "Q0_5" : Bool AT %DB2.DBX4.5, 100 ms
   "Q0_6" : Bool AT %DB2.DBX4.6, 100 ms
   "Q0_7" : Bool AT %DB2.DBX4.7, 100 ms
   "Q1_0" : Bool AT %DB2.DBX5.0, 100 ms
   "Q1_1" : Bool AT %DB2.DBX5.1, 100 ms
   "Q1_2" : Bool AT %DB2.DBX5.2, 100 ms
   "Q1_3" : Bool AT %DB2.DBX5.3, 100 ms
   "Q1_4" : Bool AT %DB2.DBX5.4, 100 ms
   "Q1_5" : Bool AT %DB2.DBX5.5, 100 ms
   "Q1_6" : Bool AT %DB2.DBX5.6, 100 ms
   "Q1_7" : Bool AT %DB2.DBX5.7, 100 ms
   "Q70_0" : Bool AT %DB2.DBX6.0, 100 ms
   "Q70_1" : Bool AT %DB2.DBX6.1, 100 ms
   "Q70_2" : Bool AT %DB2.DBX6.2, 100 ms
   "Q70_3" : Bool AT %DB2.DBX6.3, 100 ms
   "Q70_4" : Bool AT %DB2.DBX6.4, 100 ms
   "Q70_5" : Bool AT %DB2.DBX6.5, 100 ms
   "Q70_6" : Bool AT %DB2.DBX6.6, 100 ms
   "Q70_7" : Bool AT %DB2.DBX6.7, 100 ms
   "Q71_0" : Bool AT %DB2.DBX7.0, 100 ms
   "Q71_1" : Bool AT %DB2.DBX7.1, 100 ms
   "Q71_2" : Bool AT %DB2.DBX7.2, 100 ms
   "Q71_3" : Bool AT %DB2.DBX7.3, 100 ms
   "Q71_4" : Bool AT %DB2.DBX7.4, 100 ms
   "Q71_5" : Bool AT %DB2.DBX7.5, 100 ms
   "Q71_6" : Bool AT %DB2.DBX7.6, 100 ms
   "Q71_7" : Bool AT %DB2.DBX7.7, 100 ms
   "PartRelease" : Bool AT %DB2.DBX182.0, 100 ms

HMI tags "SIEMENS SIM Tags"
   "SIMPWRON" : Bool AT %DB2.DBX8.0, 100 ms
   "SIM_Divert_Animation" : DInt AT %DB2.DBD114, 100 ms
   "SIM_Lift_Animation" : DInt AT %DB2.DBD10, 100 ms
   "SIM_Reject_Animation" : DInt AT %DB2.DBD62, 100 ms

HMI tags "StringVariables"
   "String Variables_INT1_TEXT" : String[254] = PLC "String Variables".INT1_TEXT, 100 ms
   "String Variables_INT2_TEXT" : String[254] = PLC "String Variables".INT2_TEXT, 100 ms
   "String Variables_INT3_TEXT" : String[254] = PLC "String Variables".INT3_TEXT, 100 ms
   "String Variables_INT4_TEXT" : String[254] = PLC "String Variables".INT4_TEXT, 100 ms
   "String Variables_REAL1_TEXT" : String[254] = PLC "String Variables".REAL1_TEXT, 100 ms
   "String Variables_REAL2_TEXT" : String[254] = PLC "String Variables".REAL2_TEXT, 100 ms
   "String Variables_REAL3_TEXT" : String[254] = PLC "String Variables".REAL3_TEXT, 100 ms
   "String Variables_REAL4_TEXT" : String[254] = PLC "String Variables".REAL4_TEXT, 100 ms

screen "10 - PROJECT SCREEN" 480x800, template "Template"
   on GenerateScreen: SetBit("I0_1"); SetBit("SIEMENS GRAYPB")
   Button "Button_9" at 268,334 size 50x50; TextOff 'Text'; PictureOff "3-D yellow button (not pressed)"; PictureOn "3-D yellow button (pressed)"
      on Press: SetBit("I0_2")
      on Release: ResetBit("I0_2")
   Button "Button_10" at 333,334 size 50x50; TextOff 'Text'; PictureOff "3-D red button (not pressed)"; PictureOn "3-D red button (pressed)"
      on Press: SetBit("I0_3")
      on Release: ResetBit("I0_3")
   TextField "Text Field_1" at 0,0 size 480x50; Text 'SIEMENS PROJECT'
      Visibility <- "Station"
   Button "Button_1" at 53,695 size 50x50; TextOff 'Text'; PictureOff "3-D black button (not pressed)"; PictureOn "3-D black button (pressed)"
      on Press: ResetBit("SIEMENS GRAYPB")
      on Release: SetBit("SIEMENS GRAYPB")
   Button "Button_4" at 122,695 size 50x50; TextOff 'Text'; PictureOff "3-D blue button (not pressed)"; PictureOn "3-D blue button (pressed)"
      on Press: SetBit("SIEMENS BLUEPB")
      on Release: ResetBit("SIEMENS BLUEPB")
   Button "Button_6" at 192,695 size 50x50; TextOff 'Text'; PictureOff "3-D green button (not pressed)"; PictureOn "3-D green button (pressed)"
      on Press: SetBit("SIEMENS GREENPB")
      on Release: ResetBit("SIEMENS GREENPB")
   Circle "Circle_2" at 200,651 size 40x40
      Appearance <- "SIEMENS GREENLT"
   Circle "Circle_3" at 130,651 size 40x40
      Appearance <- "SIEMENS BLUELT"
   Circle "Circle_4" at 61,651 size 40x40
      Appearance <- "SIEMENS GRAYLT"
   Circle "Circle_1" at 269,651 size 40x40
      Appearance <- "SIEMENS YELLOWLT"
   TextField "Text Field_4" at 38,626 size 100x20; Text 'TP.PLC.GRAY.LT'
   TextField "Text Field_8" at 103,626 size 100x20; Text 'TP.PLC.BLUE.LT'
   TextField "Text Field_9" at 173,626 size 100x20; Text 'TP.PLC.GREEN.LT'
   TextField "Text Field_10" at 247,626 size 100x20; Text 'TP.PLC.YELLOW.LT'
   Circle "Circle_5" at 339,651 size 40x40
      Appearance <- "SIEMENS REDLT"
   TextField "Text Field_11" at 316,626 size 100x20; Text 'TP.PLC.RED.LT'
   TextField "Text Field_5" at 33,756 size 100x35; Text 'TP.PLC.GREY.PB (NC)'
   TextField "Text Field_13" at 103,756 size 100x35; Text 'TP.PLC.BLUE.PB (NO)'
   TextField "Text Field_14" at 168,756 size 100x35; Text 'TP.PLC.GREEN.PB (NO)'
   TextField "Text Field_15" at 242,756 size 100x35; Text 'TP.PLC.YELLOW.PB'
   TextField "Text Field_16" at 311,756 size 100x35; Text 'TP.PLC.RED.PB'
   IOField "IO Field_1" at 124,528 size 80x22; FormatPattern 9999
      ProcessValue <- "SIEMENS INT2"
   IOField "IO Field_3" at 124,560 size 80x22; FormatPattern 9999
      ProcessValue <- "SIEMENS INT3"
   IOField "IO Field_4" at 124,592 size 80x22; FormatPattern 9999
      ProcessValue <- "SIEMENS INT4"
   IOField "IO Field_9" at 320,528 size 80x22; FormatPattern 9999.99
      ProcessValue <- "SIEMENS REAL2"
   IOField "IO Field_10" at 320,560 size 80x22; FormatPattern 9999.99
      ProcessValue <- "SIEMENS REAL3"
   IOField "IO Field_11" at 320,592 size 80x22; FormatPattern 9999.99
      ProcessValue <- "SIEMENS REAL4"
   Switch "Switch_1" at 331,695 size 50x50; TextOn '1'; TextOff '0'; CaptionText 'Switch'; PictureOff "3-D red button (not pressed)"; PictureOn "3-D red button (pressed)"
      ProcessValue <- "SIEMENS REDPB"
   Switch "Switch_2" at 261,695 size 50x50; TextOn '1'; TextOff '0'; CaptionText 'Switch'; PictureOff "3-D yellow button (not pressed)"; PictureOn "3-D yellow button (pressed)"
      ProcessValue <- "SIEMENS YELLOWPB"
   IOField "IO Field_2" at 124,497 size 80x22; FormatPattern 9999
      ProcessValue <- "SIEMENS INT1"
   IOField "IO Field_5" at 320,497 size 80x22; FormatPattern 9999.99
      ProcessValue <- "SIEMENS REAL1"
   Button "Button_2" at 131,331 size 50x50; TextOff 'Text'; PictureOff "3-D green button (not pressed)"; PictureOn "3-D green button (pressed)"
      on Press: SetBit("SIMPWRON")
      on Release: ResetBit("SIMPWRON")
   Button "Button_3" at 201,334 size 50x50; TextOff 'Text'; PictureOff "3-D green button (not pressed)"; PictureOn "3-D green button (pressed)"
      on Press: SetBit("I0_0")
      on Release: ResetBit("I0_0")
   Button "Button_5" at 201,392 size 50x50; TextOff 'Text'; PictureOff "3-D black button (not pressed)"; PictureOn "3-D black button (pressed)"
      on Press: ResetBit("I0_1")
      on Release: SetBit("I0_1")
   TextField "Text Field_2" at 32,282 size 100x44; Text 'ESTOP PB I0.6'
   TextField "Text Field_21" at 105,282 size 100x44; Text 'POWER ON I0.5'
   TextField "Text Field_22" at 182,282 size 100x44; Text 'START PB I0.0 LT Q0.0'
   TextField "Text Field_23" at 251,282 size 100x44; Text 'PBA PB I0.2 LT Q0.2'
   TextField "Text Field_24" at 314,282 size 100x44; Text 'PBB PB I0.3 LT Q0.3'
   TextField "Text Field_25" at 173,445 size 100x44; Text 'STOP PB I0.1'
   TextField "Text Field_26" at 104,444 size 100x44; Text 'GATE SWITCH I0.7'
   TextField "Text Field_27" at 239,442 size 100x44; Text 'SSA I0.4'
   Circle "Circle_8" at 239,324 size 25x25
      Appearance <- "Q0_0"
   Circle "Circle_6" at 169,323 size 25x25
      Appearance <- "I0_5"
   Circle "Circle_7" at 309,324 size 25x25
      Appearance <- "Q0_2"
   Circle "Circle_9" at 371,324 size 25x25
      Appearance <- "Q0_3"
   Switch "Switch_3" at 266,392 size 50x50; TextOn 'ON'; TextOff 'OFF'; CaptionText 'Switch'; PictureOff "Rotary_N_Off_mono"; PictureOn "Rotary_N_On_mono"
      ProcessValue <- "I0_4"
   Switch "Switch_4" at 131,392 size 50x50; TextOn 'ON'; TextOff 'OFF'; CaptionText 'Switch'; PictureOff "Rotary_N_Off_mono"; PictureOn "Rotary_N_On_mono"
      ProcessValue <- "I0_7"
   Switch "Switch_5" at 61,331 size 50x50; TextOn '1'; TextOff '0'; CaptionText 'Switch'; PictureOff "3-D red button (not pressed)"; PictureOn "3-D red button (pressed)"
      ProcessValue <- "I0_6"
   TextField "Text Field_49" at 105,379 size 100x18; Text 'OFF ON'
   TextField "Text Field_50" at 241,379 size 100x18; Text 'OFF ON'
   TextField "Text field_34" at 520,220 size 31x18; Text 'I0.7'
   TextField "Text field_35" at 520,107 size 31x18; Text 'I0.6'
   Rectangle "Rectangle_7" at 213,189 size 47x30
      Visibility <- "I70_5"
   Rectangle "Rectangle_2" at 213,189 size 47x10
      Visibility <- "I70_5"
   Rectangle "Rectangle_3" at 366,86 size 8x92
      VerticalMovement <- "SIM_Reject_Animation"
      Visibility <- "I70_0"
   Rectangle "Rectangle_4" at 70,100 size 183x8
      HorizontalMovement <- "SIM_Lift_Animation"
   Rectangle "Rectangle_9" at 232,93 size 21x22
      HorizontalMovement <- "SIM_Lift_Animation"
   Rectangle "Rectangle_15" at 229,179 size 24x11
      Visibility <- "I70_6"
   Rectangle "Rectangle_16" at 363,168 size 14x10
      VerticalMovement <- "SIM_Reject_Animation"
      Visibility <- "I70_0"
   Rectangle "Rectangle_18" at 358,177 size 24x11
      VerticalMovement <- "SIM_Reject_Animation"
      Visibility <- "I71_1"
   TextField "Text field_28" at 202,227 size 77x18; Text 'Reject Bin'
   TextField "Text field_29" at 339,194 size 67x50; Text 'Case'
   Rectangle "Rectangle_20" at 252,183 size 7x36
      Visibility <- "I70_5"
   Rectangle "Rectangle_19" at 238,86 size 8x92
      VerticalMovement <- "SIM_Reject_Animation"
      Visibility <- "I70_1"
   Rectangle "Rectangle_21" at 235,169 size 14x10
      VerticalMovement <- "SIM_Reject_Animation"
      Visibility <- "I70_1"
   Rectangle "Rectangle_22" at 229,179 size 24x11
      VerticalMovement <- "SIM_Reject_Animation"
      Visibility <- "I71_0"
   IOField "I/O field_1" at 78,227 size 59x23; FormatPattern 99999
      ProcessValue <- "SIEMENS CH0"
   TextField "Text field_30" at 45,209 size 117x18; Text 'WEIGHT SENSOR'
   Circle "Circle_10" at 97,109 size 11x11
      Appearance <- "Q70_2"
   TextField "Text field_31" at 108,107 size 67x14; Text 'RAISE Q70.2'
   Circle "Circle_11" at 97,120 size 11x11
      Appearance <- "Q70_3"
   TextField "Text field_32" at 108,118 size 72x14; Text 'LOWER Q70.3'
   Circle "Circle_14" at 97,77 size 11x11
      Appearance <- "Q70_0"
   TextField "Text field_42" at 108,75 size 55x14; Text 'EXT Q70.0'
   Circle "Circle_12" at 97,89 size 11x11
      Appearance <- "Q70_1"
   TextField "Text field_33" at 108,87 size 56x14; Text 'RET Q70.1'
   Circle "Circle_13" at 97,132 size 11x11
      Appearance <- "Q70_4"
   TextField "Text field_36" at 108,130 size 62x14; Text 'GRIP Q70.4'
   Circle "Circle_15" at 261,204 size 11x11
      Appearance <- "Q70_5"
   TextField "Text field_37" at 272,202 size 55x14; Text 'EXT Q70.5'
   Rectangle "Rectangle_23" at 383,107 size 6x10
      Appearance <- "I70_2"
   Rectangle "Rectangle_24" at 385,160 size 6x10
      Appearance <- "I70_3"
   TextField "Text field_38" at 387,105 size 72x14; Text 'RAISED I70.2'
   TextField "Text field_39" at 389,158 size 67x14; Text 'LWR'D I70.3'
   Rectangle "Rectangle_25" at 365,76 size 10x6
      Appearance <- "I70_0"
   Rectangle "Rectangle_26" at 237,76 size 10x6
      Appearance <- "I70_1"
   TextField "Text field_40" at 339,61 size 63x14; Text 'EXT'D I70.0'
   TextField "Text field_41" at 210,61 size 64x14; Text 'RET'D I70.1'
   Button "Button_7" at 256,139 size 53x35; TextOff 'CLEAR/SET PART AT PICKUP'
      on Press: InvertBit("I70_6")
   Rectangle "Rectangle_27" at 261,185 size 6x10
      Appearance <- "I70_5"
   TextField "Text field_43" at 265,183 size 64x14; Text 'RET'D I70.5'
   Rectangle "Rectangle_28" at 201,166 size 28x8
      Appearance <- "I70_6"
   TextField "Text field_45" at 193,132 size 41x26; Text 'PART AT PICKUP'
   TextField "Text field_46" at 200,153 size 32x14; Text 'I70.6'
   Circle "Circle_16" at 35,166 size 11x11
      Appearance <- "Q70_6"
   TextField "Text field_44" at 46,164 size 58x14; Text 'RUN Q70.6'
   TextField "Text field_47" at 45,227 size 31x18; Text 'IW2'
   Rectangle "Rectangle_29" at 229,194 size 24x21
      Visibility <- "I70_5"
   IOField "I/O field_15" at 217,584 size 96x36; FormatPattern ????????????
      ProcessValue <- "String Variables_REAL4_TEXT"
   IOField "I/O field_19" at 21,583 size 96x36; FormatPattern ????????????
      ProcessValue <- "String Variables_INT4_TEXT"
   IOField "I/O field_12" at 217,492 size 96x36; FormatPattern ????????????
      ProcessValue <- "String Variables_REAL1_TEXT"
   IOField "I/O field_13" at 217,521 size 96x36; FormatPattern ????????????
      ProcessValue <- "String Variables_REAL2_TEXT"
   IOField "I/O field_14" at 217,551 size 96x36; FormatPattern ????????????
      ProcessValue <- "String Variables_REAL3_TEXT"
   IOField "I/O field_16" at 21,491 size 96x36; FormatPattern ????????????
      ProcessValue <- "String Variables_INT1_TEXT"
   IOField "I/O field_17" at 21,520 size 96x36; FormatPattern ????????????
      ProcessValue <- "String Variables_INT2_TEXT"
   IOField "I/O field_18" at 21,550 size 96x36; FormatPattern ????????????
      ProcessValue <- "String Variables_INT3_TEXT"

screen "00 - A2148 LAB SIMULATOR" 480x800, template "Template"
   on GenerateScreen: SetBit("I0_1"); SetBit("SIEMENS GRAYPB")
   Rectangle "Rectangle_3" at 345,125 size 35x30
      VerticalMovement <- "SIM_Lift_Animation"
   Button "Button_9" at 268,334 size 50x50; TextOff 'Text'; PictureOff "3-D yellow button (not pressed)"; PictureOn "3-D yellow button (pressed)"
      on Press: SetBit("I0_2")
      on Release: ResetBit("I0_2")
   Button "Button_10" at 333,334 size 50x50; TextOff 'Text'; PictureOff "3-D red button (not pressed)"; PictureOn "3-D red button (pressed)"
      on Press: SetBit("I0_3")
      on Release: ResetBit("I0_3")
   TextField "Text Field_1" at 0,0 size 480x50; Text 'A2148 SIEMENS LAB SIMULATOR'
      Visibility <- "Station"
   Button "Button_1" at 53,695 size 50x50; TextOff 'Text'; PictureOff "3-D black button (not pressed)"; PictureOn "3-D black button (pressed)"
      on Press: ResetBit("SIEMENS GRAYPB")
      on Release: SetBit("SIEMENS GRAYPB")
   Button "Button_4" at 122,695 size 50x50; TextOff 'Text'; PictureOff "3-D blue button (not pressed)"; PictureOn "3-D blue button (pressed)"
      on Press: SetBit("SIEMENS BLUEPB")
      on Release: ResetBit("SIEMENS BLUEPB")
   Button "Button_6" at 192,695 size 50x50; TextOff 'Text'; PictureOff "3-D green button (not pressed)"; PictureOn "3-D green button (pressed)"
      on Press: SetBit("SIEMENS GREENPB")
      on Release: ResetBit("SIEMENS GREENPB")
   Circle "Circle_2" at 200,651 size 40x40
      Appearance <- "SIEMENS GREENLT"
   Circle "Circle_3" at 130,651 size 40x40
      Appearance <- "SIEMENS BLUELT"
   Circle "Circle_4" at 61,651 size 40x40
      Appearance <- "SIEMENS GRAYLT"
   Circle "Circle_1" at 269,651 size 40x40
      Appearance <- "SIEMENS YELLOWLT"
   TextField "Text Field_4" at 38,626 size 100x20; Text 'TP.PLC.GRAY.LT'
   TextField "Text Field_8" at 103,626 size 100x20; Text 'TP.PLC.BLUE.LT'
   TextField "Text Field_9" at 173,626 size 100x20; Text 'TP.PLC.GREEN.LT'
   TextField "Text Field_10" at 247,626 size 100x20; Text 'TP.PLC.YELLOW.LT'
   Circle "Circle_5" at 339,651 size 40x40
      Appearance <- "SIEMENS REDLT"
   TextField "Text Field_11" at 316,626 size 100x20; Text 'TP.PLC.RED.LT'
   TextField "Text Field_5" at 33,756 size 100x35; Text 'TP.PLC.GREY.PB (NC)'
   TextField "Text Field_13" at 103,756 size 100x35; Text 'TP.PLC.BLUE.PB (NO)'
   TextField "Text Field_14" at 168,756 size 100x35; Text 'TP.PLC.GREEN.PB (NO)'
   TextField "Text Field_15" at 242,756 size 100x35; Text 'TP.PLC.YELLOW.PB'
   TextField "Text Field_16" at 311,756 size 100x35; Text 'TP.PLC.RED.PB'
   IOField "IO Field_1" at 124,528 size 80x22; FormatPattern 9999
      ProcessValue <- "SIEMENS INT2"
   TextField "Text Field_3" at 13,499 size 100x20; Text 'TP.PLC.INT1'
   TextField "Text Field_6" at 16,530 size 100x20; Text 'TP.PLC.INT2'
   IOField "IO Field_3" at 124,560 size 80x22; FormatPattern 9999
      ProcessValue <- "SIEMENS INT3"
   TextField "Text Field_7" at 16,562 size 100x20; Text 'TP.PLC.INT3'
   IOField "IO Field_4" at 124,592 size 80x22; FormatPattern 9999
      ProcessValue <- "SIEMENS INT4"
   TextField "Text Field_12" at 16,594 size 100x20; Text 'TP.PLC.INT4'
   TextField "Text Field_17" at 211,499 size 100x20; Text 'TP.PLC.REAL1'
   TextField "Text Field_18" at 214,530 size 100x20; Text 'TP.PLC.REAL2'
   TextField "Text Field_19" at 214,562 size 100x20; Text 'TP.PLC.REAL3'
   TextField "Text Field_20" at 214,594 size 100x20; Text 'TP.PLC.REAL4'
   IOField "IO Field_9" at 320,528 size 80x22; FormatPattern 9999.99
      ProcessValue <- "SIEMENS REAL2"
   IOField "IO Field_10" at 320,560 size 80x22; FormatPattern 9999.99
      ProcessValue <- "SIEMENS REAL3"
   IOField "IO Field_11" at 320,592 size 80x22; FormatPattern 9999.99
      ProcessValue <- "SIEMENS REAL4"
   Switch "Switch_1" at 331,695 size 50x50; TextOn '1'; TextOff '0'; CaptionText 'Switch'; PictureOff "3-D red button (not pressed)"; PictureOn "3-D red button (pressed)"
      ProcessValue <- "SIEMENS REDPB"
   Switch "Switch_2" at 261,695 size 50x50; TextOn '1'; TextOff '0'; CaptionText 'Switch'; PictureOff "3-D yellow button (not pressed)"; PictureOn "3-D yellow button (pressed)"
      ProcessValue <- "SIEMENS YELLOWPB"
   IOField "IO Field_2" at 124,497 size 80x22; FormatPattern 9999
      ProcessValue <- "SIEMENS INT1"
   IOField "IO Field_5" at 320,497 size 80x22; FormatPattern 9999.99
      ProcessValue <- "SIEMENS REAL1"
   Button "Button_2" at 131,331 size 50x50; TextOff 'Text'; PictureOff "3-D green button (not pressed)"; PictureOn "3-D green button (pressed)"
      on Press: SetBit("SIMPWRON")
      on Release: ResetBit("SIMPWRON")
   Button "Button_3" at 201,334 size 50x50; TextOff 'Text'; PictureOff "3-D green button (not pressed)"; PictureOn "3-D green button (pressed)"
      on Press: SetBit("I0_0")
      on Release: ResetBit("I0_0")
   Button "Button_5" at 201,392 size 50x50; TextOff 'Text'; PictureOff "3-D black button (not pressed)"; PictureOn "3-D black button (pressed)"
      on Press: ResetBit("I0_1")
      on Release: SetBit("I0_1")
   TextField "Text Field_2" at 32,282 size 100x44; Text 'ESTOP PB I0.6'
   TextField "Text Field_21" at 105,282 size 100x44; Text 'POWER ON I0.5'
   TextField "Text Field_22" at 182,282 size 100x44; Text 'START PB I0.0 LT Q0.0'
   TextField "Text Field_23" at 251,282 size 100x44; Text 'PBA PB I0.2 LT Q0.2'
   TextField "Text Field_24" at 314,282 size 100x44; Text 'PBB PB I0.3 LT Q0.3'
   TextField "Text Field_25" at 173,445 size 100x44; Text 'STOP PB I0.1'
   TextField "Text Field_26" at 104,444 size 100x44; Text 'GATE SWITCH I0.7'
   TextField "Text Field_27" at 239,442 size 100x44; Text 'SSA I0.4'
   Circle "Circle_8" at 239,324 size 25x25
      Appearance <- "Q0_0"
   Circle "Circle_6" at 169,323 size 25x25
      Appearance <- "I0_5"
   Circle "Circle_7" at 309,324 size 25x25
      Appearance <- "Q0_2"
   Circle "Circle_9" at 371,324 size 25x25
      Appearance <- "Q0_3"
   Rectangle "Rectangle_4" at 377,125 size 6x30
      VerticalMovement <- "SIM_Lift_Animation"
   Rectangle "Rectangle_8" at 296,166 size 4x20
      Visibility <- "PartRelease"
   Rectangle "Rectangle_10" at 219,177 size 8x34
      VerticalMovement <- "SIM_Reject_Animation"
   Polygon "Polygon_1" at 219,174 size 39x3
      VerticalMovement <- "SIM_Reject_Animation"
   Rectangle "Rectangle_15" at 330,165 size 4x20
      Visibility <- "PartRelease"
   Rectangle "Rectangle_17" at 156,177 size 8x34
      VerticalMovement <- "SIM_Divert_Animation"
   Polygon "Polygon_3" at 156,174 size 39x3
      VerticalMovement <- "SIM_Divert_Animation"
   Circle "Circle_10" at 348,110 size 11x11
      Appearance <- "Q70_0"
   TextField "Text field_28" at 359,108 size 67x14; Text 'RAISE Q70.0'
   Circle "Circle_11" at 348,98 size 11x11
      Appearance <- "Q70_1"
   TextField "Text field_29" at 359,96 size 72x14; Text 'LOWER Q70.1'
   Rectangle "Rectangle_6" at 383,125 size 6x10
      Appearance <- "I70_1"
   Rectangle "Rectangle_11" at 383,145 size 6x10
      Appearance <- "I70_0"
   TextField "Text field_30" at 387,123 size 32x14; Text 'I70.1'
   TextField "Text field_31" at 387,143 size 32x14; Text 'I70.0'
   TextField "Text field_32" at 390,132 size 33x15; Text 'LIFT'
   TextField "Text field_33" at 339,173 size 94x15; Text 'PART RELEASE'
   Circle "Circle_12" at 343,187 size 11x11
      Appearance <- "Q70_6"
   TextField "Text field_34" at 354,185 size 56x14; Text 'REL Q70.6'
   TextField "Text field_35" at 226,175 size 49x15; Text 'REJECT'
   TextField "Text field_36" at 162,175 size 50x15; Text 'DIVERT'
   Rectangle "Rectangle_12" at 232,188 size 6x10
      Appearance <- "I70_2"
   Rectangle "Rectangle_18" at 232,225 size 6x10
      Appearance <- "I70_3"
   TextField "Text field_37" at 236,186 size 32x14; Text 'I70.2'
   TextField "Text field_38" at 236,223 size 32x14; Text 'I70.3'
   Circle "Circle_13" at 216,236 size 11x11
      Appearance <- "Q70_2"
   TextField "Text field_39" at 227,234 size 55x14; Text 'EXT Q70.2'
   Rectangle "Rectangle_19" at 169,188 size 6x10
      Appearance <- "I70_4"
   Rectangle "Rectangle_20" at 169,225 size 6x10
      Appearance <- "I70_5"
   TextField "Text field_40" at 173,186 size 32x14; Text 'I70.4'
   TextField "Text field_41" at 173,223 size 32x14; Text 'I70.5'
   Circle "Circle_14" at 153,236 size 11x11
      Appearance <- "Q70_4"
   TextField "Text field_42" at 164,234 size 55x14; Text 'EXT Q70.4'
   Rectangle "Rectangle_21" at 310,175 size 9x20
      Appearance <- "I71_0"
   TextField "Text field_43" at 302,195 size 32x14; Text 'I71.0'
   TextField "Text field_44" at 293,204 size 72x26; Text 'PART AT RELEASE'
   Rectangle "Rectangle_22" at 303,112 size 28x8
      Appearance <- "I71_1"
   TextField "Text field_45" at 265,78 size 102x26; Text 'PART MOVING ONTO LIFT'
   TextField "Text field_46" at 302,99 size 32x14; Text 'I71.1'
   IOField "IO Field_6" at 242,105 size 36x13; FormatPattern s99999
      ProcessValue <- "SIEMENS CH0"
   TextField "Text field_47" at 247,92 size 24x14; Text 'CH0'
   TextField "Text field_48" at 164,91 size 93x15; Text 'PART HEIGHT'
   Rectangle "Rectangle_23" at 300,160 size 30x13
      Appearance <- "I71_0"
   Circle "Circle_16" at 303,124 size 30x30
      Appearance <- "I71_1"
   Button "Button_7" at 309,230 size 98x34; TextOff 'CLEAR/SET PART AT PART RELEASE'
      on Press: InvertBit("I71_0")
   Button "Button_8" at 302,44 size 98x34; TextOff 'CLEAR/SET PART ON CONVEYOR'
      on Press: InvertBit("I71_1")
   Switch "Switch_3" at 266,392 size 50x50; TextOn 'ON'; TextOff 'OFF'; CaptionText 'Switch'; PictureOff "Rotary_N_Off_mono"; PictureOn "Rotary_N_On_mono"
      ProcessValue <- "I0_4"
   Switch "Switch_4" at 131,392 size 50x50; TextOn 'ON'; TextOff 'OFF'; CaptionText 'Switch'; PictureOff "Rotary_N_Off_mono"; PictureOn "Rotary_N_On_mono"
      ProcessValue <- "I0_7"
   Switch "Switch_5" at 61,331 size 50x50; TextOn '1'; TextOff '0'; CaptionText 'Switch'; PictureOff "3-D red button (not pressed)"; PictureOn "3-D red button (pressed)"
      ProcessValue <- "I0_6"
   TextField "Text Field_49" at 105,379 size 100x18; Text 'OFF ON'
   TextField "Text Field_50" at 241,379 size 100x18; Text 'OFF ON'
*)